LIN {X 0,Y 228.814,Z 416.35,A -85,B 0,C 180,E1 -20899.749,E2 -20899.749} C_VEL
LIN {X 0,Y 233.33,Z 413.266,A -85,B 0,C 180,E1 -20902.12,E2 -20902.12} C_VEL
LIN {X 0,Y 238.29,Z 408.992,A -85,B 0,C 180,E1 -20904.39,E2 -20904.39} C_VEL
LIN {X 0,Y 239.683,Z 407.452,A -85,B 0,C 180,E1 -20905.163,E2 -20905.163} C_VEL
LIN {X 0,Y 241.807,Z 403.361,A -85,B 0,C 180,E1 -20907.714,E2 -20907.714} C_VEL
LIN {X 0,Y 243.168,Z 399.95,A -85,B 0,C 180,E1 -20909.882,E2 -20909.882} C_VEL
LIN {X 0,Y 244.629,Z 395.449,A -85,B 0,C 180,E1 -20913.085,E2 -20913.085} C_VEL
LIN {X 0,Y 245.074,Z 393.5,A -85,B 0,C 180,E1 -20915,E2 -20915} C_VEL
LIN {X 0,Y 245.23,Z 392.181,A -85,B 0,C 180,E1 -20917.004,E2 -20917.004} C_VEL
LIN {X 0,Y 245.282,Z 391.515,A -85,B 0,C 180,E1 -20919.319,E2 -20919.319} C_VEL
LIN {X 0,Y 245.496,Z 391.651,A -85,B 0,C 180,E1 -20921.899,E2 -20921.899} C_VEL
LIN {X 0,Y 245.947,Z 392.643,A -85,B 0,C 180,E1 -20924.407,E2 -20924.407} C_VEL
LIN {X 0,Y 246.92,Z 395.234,A -85,B 0,C 180,E1 -20927.736,E2 -20927.736} C_VEL
LIN {X 0,Y 247.592,Z 398.254,A -85,B 0,C 180,E1 -20930.035,E2 -20930.035} C_VEL
LIN {X 0,Y 247.879,Z 400.529,A -85,B 0,C 180,E1 -20931.409,E2 -20931.409} C_VEL
LIN {X 0,Y 247.014,Z 403.447,A -85,B 0,C 180,E1 -20932.402,E2 -20932.402} C_VEL
LIN {X 0,Y 243.965,Z 411.2,A -85,B 0,C 180,E1 -20934.82,E2 -20934.82} C_VEL
LIN {X 0,Y 240.711,Z 417.71,A -85,B 0,C 180,E1 -20936.808,E2 -20936.808} C_VEL
LIN {X 0,Y 236.558,Z 423.872,A -85,B 0,C 180,E1 -20938.673,E2 -20938.673} C_VEL
LIN {X 0,Y 231.251,Z 430.368,A -85,B 0,C 180,E1 -20940.905,E2 -20940.905} C_VEL
LIN {X 0,Y 225.202,Z 437.275,A -85,B 0,C 180,E1 -20944.093,E2 -20944.093} C_VEL
LIN {X 0,Y 222.213,Z 440.446,A -85,B 0,C 180,E1 -20946.02,E2 -20946.02} C_VEL
LIN {X 0,Y 219.813,Z 442.378,A -85,B 0,C 180,E1 -20947.335,E2 -20947.335} C_VEL
LIN {X 0,Y 214.43,Z 444.919,A -85,B 0,C 180,E1 -20949.437,E2 -20949.437} C_VEL
LIN {X 0,Y 209.432,Z 446.66,A -85,B 0,C 180,E1 -20951.695,E2 -20951.695} C_VEL
LIN {X 0,Y 207.679,Z 447.347,A -85,B 0,C 180,E1 -20953.224,E2 -20953.224} C_VEL
LIN {X 0,Y 206.133,Z 448.199,A -85,B 0,C 180,E1 -20956.192,E2 -20956.192} C_VEL
LIN {X 0,Y 205.327,Z 448.115,A -85,B 0,C 180,E1 -20960.146,E2 -20960.146} C_VEL
LIN {X 0,Y 205.557,Z 446.587,A -85,B 0,C 180,E1 -20964.113,E2 -20964.113} C_VEL
LIN {X 0,Y 206.007,Z 445.284,A -85,B 0,C 180,E1 -20966.088,E2 -20966.088} C_VEL
LIN {X 0,Y 206.791,Z 442.454,A -85,B 0,C 180,E1 -20969.026,E2 -20969.026} C_VEL
LIN {X 0,Y 207.458,Z 438.737,A -85,B 0,C 180,E1 -20971.881,E2 -20971.881} C_VEL
LIN {X 0,Y 206.568,Z 441.761,A -85,B 0,C 180,E1 -20973.902,E2 -20973.902} C_VEL
LIN {X 0,Y 205.939,Z 443.935,A -85,B 0,C 180,E1 -20975.876,E2 -20975.876} C_VEL
LIN {X 0,Y 205.61,Z 445.513,A -85,B 0,C 180,E1 -20977.858,E2 -20977.858} C_VEL
LIN {X 0,Y 205.582,Z 446.527,A -85,B 0,C 180,E1 -20979.842,E2 -20979.842} C_VEL
LIN {X 0,Y 205.912,Z 446.997,A -85,B 0,C 180,E1 -20981.817,E2 -20981.817} C_VEL
LIN {X 0,Y 206.627,Z 446.963,A -85,B 0,C 180,E1 -20983.774,E2 -20983.774} C_VEL
LIN {X 0,Y 207.622,Z 446.402,A -85,B 0,C 180,E1 -20985.712,E2 -20985.712} C_VEL
LIN {X 0,Y 209.104,Z 445.335,A -85,B 0,C 180,E1 -20987.607,E2 -20987.607} C_VEL
LIN {X 0,Y 211.961,Z 442.735,A -85,B 0,C 180,E1 -20990.374,E2 -20990.374} C_VEL
LIN {X 0,Y 215.478,Z 438.804,A -85,B 0,C 180,E1 -20993.041,E2 -20993.041} C_VEL
LIN {X 0,Y 219.824,Z 433.439,A -85,B 0,C 180,E1 -20995.57,E2 -20995.57} C_VEL
LIN {X 0,Y 223.914,Z 427.641,A -85,B 0,C 180,E1 -20997.578,E2 -20997.578} C_VEL
LIN {X 0,Y 228.592,Z 420.356,A -85,B 0,C 180,E1 -20999.467,E2 -20999.467} C_VEL
LIN {X 0,Y 232.382,Z 412.031,A -85,B 0,C 180,E1 -21001.4,E2 -21001.4} C_VEL
LIN {X 0,Y 233.877,Z 408.212,A -85,B 0,C 180,E1 -21002.188,E2 -21002.188} C_VEL
LIN {X 0,Y 235.674,Z 399.15,A -85,B 0,C 180,E1 -21004.513,E2 -21004.513} C_VEL
LIN {X 0,Y 236.749,Z 389.553,A -85,B 0,C 180,E1 -21007.182,E2 -21007.182} C_VEL
LIN {X 0,Y 236.748,Z 388.634,A -85,B 0,C 180,E1 -21007.486,E2 -21007.486} C_VEL
LIN {X 0,Y 236.034,Z 385.627,A -85,B 0,C 180,E1 -21009.268,E2 -21009.268} C_VEL
LIN {X 0,Y 235.075,Z 383.096,A -85,B 0,C 180,E1 -21011.63,E2 -21011.63} C_VEL
LIN {X 0,Y 234.344,Z 381.808,A -85,B 0,C 180,E1 -21013.963,E2 -21013.963} C_VEL
LIN {X 0,Y 233.881,Z 381.582,A -85,B 0,C 180,E1 -21016.277,E2 -21016.277} C_VEL
LIN {X 0,Y 233.809,Z 382.151,A -85,B 0,C 180,E1 -21018.718,E2 -21018.718} C_VEL
LIN {X 0,Y 234.028,Z 383.771,A -85,B 0,C 180,E1 -21021.334,E2 -21021.334} C_VEL
LIN {X 0,Y 234.447,Z 385.325,A -85,B 0,C 180,E1 -21023.161,E2 -21023.161} C_VEL
LIN {X 0,Y 234.718,Z 388.125,A -85,B 0,C 180,E1 -21025.324,E2 -21025.324} C_VEL
LIN {X 0,Y 234.45,Z 392.693,A -85,B 0,C 180,E1 -21027.833,E2 -21027.833} C_VEL
LIN {X 0,Y 233.699,Z 398.365,A -85,B 0,C 180,E1 -21030.705,E2 -21030.705} C_VEL
LIN {X 0,Y 232.609,Z 403.003,A -85,B 0,C 180,E1 -21033.048,E2 -21033.048} C_VEL
LIN {X 0,Y 231.392,Z 406.408,A -85,B 0,C 180,E1 -21034.833,E2 -21034.833} C_VEL
LIN {X 0,Y 230.175,Z 408.313,A -85,B 0,C 180,E1 -21035.655,E2 -21035.655} C_VEL
LIN {X 0,Y 225.28,Z 413.35,A -85,B 0,C 180,E1 -21038.013,E2 -21038.013} C_VEL
LIN {X 0,Y 222.294,Z 415.749,A -85,B 0,C 180,E1 -21039.647,E2 -21039.647} C_VEL
LIN {X 0,Y 219.533,Z 417.471,A -85,B 0,C 180,E1 -21041.327,E2 -21041.327} C_VEL
LIN {X 0,Y 216.997,Z 418.533,A -85,B 0,C 180,E1 -21043.051,E2 -21043.051} C_VEL
LIN {X 0,Y 214.633,Z 418.98,A -85,B 0,C 180,E1 -21044.812,E2 -21044.812} C_VEL
LIN {X 0,Y 212.473,Z 418.818,A -85,B 0,C 180,E1 -21046.61,E2 -21046.61} C_VEL
LIN {X 0,Y 210.527,Z 418.027,A -85,B 0,C 180,E1 -21048.443,E2 -21048.443} C_VEL
LIN {X 0,Y 208.193,Z 415.631,A -85,B 0,C 180,E1 -21051.26,E2 -21051.26} C_VEL
LIN {X 0,Y 206.472,Z 411.79,A -85,B 0,C 180,E1 -21054.137,E2 -21054.137} C_VEL
LIN {X 0,Y 205.572,Z 406.34,A -85,B 0,C 180,E1 -21057.058,E2 -21057.058} C_VEL
LIN {X 0,Y 205.271,Z 400.286,A -85,B 0,C 180,E1 -21059.507,E2 -21059.507} C_VEL
LIN {X 0,Y 205.338,Z 392.617,A -85,B 0,C 180,E1 -21061.959,E2 -21061.959} C_VEL
LIN {X 0,Y 205.793,Z 383.712,A -85,B 0,C 180,E1 -21064.159,E2 -21064.159} C_VEL
LIN {X 0,Y 206.062,Z 376.071,A -85,B 0,C 180,E1 -21065.625,E2 -21065.625} C_VEL
LIN {X 0,Y 206.367,Z 365.456,A -85,B 0,C 180,E1 -21067.212,E2 -21067.212} C_VEL
LIN {X 0,Y 206.597,Z 356.563,A -85,B 0,C 180,E1 -21068.221,E2 -21068.221} C_VEL
LIN {X 0,Y 205.887,Z 341.814,A -85,B 0,C 180,E1 -21076.475,E2 -21076.475} C_VEL
LIN {X 0,Y 206.128,Z 333.911,A -85,B 0,C 180,E1 -21080.975,E2 -21080.975} C_VEL
LIN {X 0,Y 206.537,Z 324.736,A -85,B 0,C 180,E1 -21086.252,E2 -21086.252} C_VEL
LIN {X 0,Y 206.884,Z 318.714,A -85,B 0,C 180,E1 -21089.787,E2 -21089.787} C_VEL
LIN {X 0,Y 206.754,Z 318.73,A -85,B 0,C 180,E1 -21092.944,E2 -21092.944} C_VEL
LIN {X 0,Y 206.669,Z 318.74,A -85,B 0,C 180,E1 -21097.739,E2 -21097.739} C_VEL
LIN {X 0,Y 206.628,Z 318.743,A -85,B 0,C 180,E1 -21101.558,E2 -21101.558} C_VEL
LIN {X 0,Y 206.624,Z 318.746,A -85,B 0,C 180,E1 -21105.58,E2 -21105.58} C_VEL
LIN {X 0,Y 206.652,Z 318.74,A -85,B 0,C 180,E1 -21109.747,E2 -21109.747} C_VEL
LIN {X 0,Y 206.691,Z 318.739,A -85,B 0,C 180,E1 -21114.687,E2 -21114.687} C_VEL
LIN {X 0,Y 206.714,Z 318.731,A -85,B 0,C 180,E1 -21119.337,E2 -21119.337} C_VEL
LIN {X 0,Y 206.724,Z 318.733,A -85,B 0,C 180,E1 -21123.771,E2 -21123.771} C_VEL
LIN {X 0,Y 206.749,Z 318.728,A -85,B 0,C 180,E1 -21128.042,E2 -21128.042} C_VEL
LIN {X 0,Y 206.867,Z 318.717,A -85,B 0,C 180,E1 -21132.196,E2 -21132.196} C_VEL
LIN {X 0,Y 206.88,Z 318.713,A -85,B 0,C 180,E1 -21136.243,E2 -21136.243} C_VEL
LIN {X 0,Y 207.069,Z 318.693,A -85,B 0,C 180,E1 -21140.229,E2 -21140.229} C_VEL
LIN {X 0,Y 207.029,Z 318.695,A -85,B 0,C 180,E1 -21144.155,E2 -21144.155} C_VEL
LIN {X 0,Y 207.334,Z 318.659,A -85,B 0,C 180,E1 -21148.057,E2 -21148.057} C_VEL
LIN {X 0,Y 207.469,Z 318.644,A -85,B 0,C 180,E1 -21150,E2 -21150} C_VEL
LIN {X 0,Y 207.334,Z 318.659,A -85,B 0,C 180,E1 -21151.943,E2 -21151.943} C_VEL
LIN {X 0,Y 207.118,Z 318.687,A -85,B 0,C 180,E1 -21157.801,E2 -21157.801} C_VEL
LIN {X 0,Y 206.91,Z 318.709,A -85,B 0,C 180,E1 -21161.759,E2 -21161.759} C_VEL
LIN {X 0,Y 206.855,Z 318.719,A -85,B 0,C 180,E1 -21165.772,E2 -21165.772} C_VEL
LIN {X 0,Y 206.803,Z 318.722,A -85,B 0,C 180,E1 -21169.867,E2 -21169.867} C_VEL
LIN {X 0,Y 206.759,Z 318.729,A -85,B 0,C 180,E1 -21174.073,E2 -21174.073} C_VEL
LIN {X 0,Y 206.735,Z 318.73,A -85,B 0,C 180,E1 -21178.42,E2 -21178.42} C_VEL
LIN {X 0,Y 206.694,Z 318.737,A -85,B 0,C 180,E1 -21182.959,E2 -21182.959} C_VEL
LIN {X 0,Y 206.672,Z 318.737,A -85,B 0,C 180,E1 -21187.742,E2 -21187.742} C_VEL
LIN {X 0,Y 206.633,Z 318.745,A -85,B 0,C 180,E1 -21191.564,E2 -21191.564} C_VEL
LIN {X 0,Y 206.624,Z 318.744,A -85,B 0,C 180,E1 -21195.585,E2 -21195.585} C_VEL
LIN {X 0,Y 206.647,Z 318.742,A -85,B 0,C 180,E1 -21199.749,E2 -21199.749} C_VEL
LIN {X 0,Y 206.783,Z 318.725,A -85,B 0,C 180,E1 -21204.709,E2 -21204.709} C_VEL
LIN {X 0,Y 207.122,Z 318.815,A -85,B 0,C 180,E1 -21208.351,E2 -21208.351} C_VEL
LIN {X 0,Y 206.657,Z 323.186,A -85,B 0,C 180,E1 -21212.155,E2 -21212.155} C_VEL
LIN {X 0,Y 206.05,Z 328.932,A -85,B 0,C 180,E1 -21217.062,E2 -21217.062} C_VEL
LIN {X 0,Y 205.493,Z 334.922,A -85,B 0,C 180,E1 -21222.076,E2 -21222.076} C_VEL
LIN {X 0,Y 205.269,Z 341.862,A -85,B 0,C 180,E1 -21227.709,E2 -21227.709} C_VEL
LIN {X 0,Y 206.4,Z 354.238,A -85,B 0,C 180,E1 -21229.085,E2 -21229.085} C_VEL
LIN {X 0,Y 206.727,Z 360.644,A -85,B 0,C 180,E1 -21229.969,E2 -21229.969} C_VEL
LIN {X 0,Y 206.197,Z 372.124,A -85,B 0,C 180,E1 -21231.924,E2 -21231.924} C_VEL
LIN {X 0,Y 205.81,Z 382.31,A -85,B 0,C 180,E1 -21234.123,E2 -21234.123} C_VEL
LIN {X 0,Y 205.337,Z 391.3,A -85,B 0,C 180,E1 -21236.569,E2 -21236.569} C_VEL
LIN {X 0,Y 205.133,Z 399.93,A -85,B 0,C 180,E1 -21239.512,E2 -21239.512} C_VEL
LIN {X 0,Y 205.32,Z 405.672,A -85,B 0,C 180,E1 -21241.964,E2 -21241.964} C_VEL
LIN {X 0,Y 206.134,Z 411.087,A -85,B 0,C 180,E1 -21244.892,E2 -21244.892} C_VEL
LIN {X 0,Y 207.525,Z 415.168,A -85,B 0,C 180,E1 -21247.788,E2 -21247.788} C_VEL
LIN {X 0,Y 208.827,Z 417.148,A -85,B 0,C 180,E1 -21249.69,E2 -21249.69} C_VEL
LIN {X 0,Y 210.385,Z 418.6,A -85,B 0,C 180,E1 -21251.565,E2 -21251.565} C_VEL
LIN {X 0,Y 212.31,Z 419.539,A -85,B 0,C 180,E1 -21253.401,E2 -21253.401} C_VEL
LIN {X 0,Y 214.482,Z 419.914,A -85,B 0,C 180,E1 -21255.199,E2 -21255.199} C_VEL
LIN {X 0,Y 216.874,Z 419.813,A -85,B 0,C 180,E1 -21256.959,E2 -21256.959} C_VEL
LIN {X 0,Y 219.491,Z 419.201,A -85,B 0,C 180,E1 -21258.677,E2 -21258.677} C_VEL
LIN {X 0,Y 222.323,Z 418.076,A -85,B 0,C 180,E1 -21260.351,E2 -21260.351} C_VEL
LIN {X 0,Y 227.004,Z 415.473,A -85,B 0,C 180,E1 -21262.77,E2 -21262.77} C_VEL
LIN {X 0,Y 232.143,Z 411.656,A -85,B 0,C 180,E1 -21265.08,E2 -21265.08} C_VEL
LIN {X 0,Y 233.739,Z 410.198,A -85,B 0,C 180,E1 -21265.85,E2 -21265.85} C_VEL
LIN {X 0,Y 236.189,Z 406.575,A -85,B 0,C 180,E1 -21268.433,E2 -21268.433} C_VEL
LIN {X 0,Y 238.124,Z 402.905,A -85,B 0,C 180,E1 -21271.139,E2 -21271.139} C_VEL
LIN {X 0,Y 239.643,Z 399.623,A -85,B 0,C 180,E1 -21273.865,E2 -21273.865} C_VEL
LIN {X 0,Y 240.137,Z 398.024,A -85,B 0,C 180,E1 -21275.829,E2 -21275.829} C_VEL
LIN {X 0,Y 240.368,Z 397.115,A -85,B 0,C 180,E1 -21277.882,E2 -21277.882} C_VEL
LIN {X 0,Y 240.641,Z 396.83,A -85,B 0,C 180,E1 -21280.594,E2 -21280.594} C_VEL
LIN {X 0,Y 241.068,Z 397.401,A -85,B 0,C 180,E1 -21283.211,E2 -21283.211} C_VEL
LIN {X 0,Y 241.771,Z 399.583,A -85,B 0,C 180,E1 -21286.615,E2 -21286.615} C_VEL
LIN {X 0,Y 242.392,Z 401.958,A -85,B 0,C 180,E1 -21288.928,E2 -21288.928} C_VEL
LIN {X 0,Y 242.593,Z 404.996,A -85,B 0,C 180,E1 -21290.942,E2 -21290.942} C_VEL
LIN {X 0,Y 239.242,Z 412.361,A -85,B 0,C 180,E1 -21293.461,E2 -21293.461} C_VEL
LIN {X 0,Y 235.819,Z 418.507,A -85,B 0,C 180,E1 -21295.511,E2 -21295.511} C_VEL
LIN {X 0,Y 231.575,Z 424.327,A -85,B 0,C 180,E1 -21297.405,E2 -21297.405} C_VEL
LIN {X 0,Y 225.149,Z 431.45,A -85,B 0,C 180,E1 -21300.037,E2 -21300.037} C_VEL
LIN {X 0,Y 218.862,Z 437.795,A -85,B 0,C 180,E1 -21303.284,E2 -21303.284} C_VEL
LIN {X 0,Y 214.916,Z 441.499,A -85,B 0,C 180,E1 -21305.873,E2 -21305.873} C_VEL
LIN {X 0,Y 211.597,Z 444.363,A -85,B 0,C 180,E1 -21308.57,E2 -21308.57} C_VEL
LIN {X 0,Y 208.267,Z 446.981,A -85,B 0,C 180,E1 -21312.32,E2 -21312.32} C_VEL
LIN {X 0,Y 207.679,Z 447.347,A -85,B 0,C 180,E1 -21313.224,E2 -21313.224} C_VEL
LIN {X 0,Y 206.148,Z 447.868,A -85,B 0,C 180,E1 -21314.798,E2 -21314.798} C_VEL
LIN {X 0,Y 202.33,Z 447.811,A -85,B 0,C 180,E1 -21317.362,E2 -21317.362} C_VEL
LIN {X 0,Y 199.528,Z 447.131,A -85,B 0,C 180,E1 -21319.475,E2 -21319.475} C_VEL
LIN {X 0,Y 198.409,Z 446.41,A -85,B 0,C 180,E1 -21321.137,E2 -21321.137} C_VEL
LIN {X 0,Y 198.339,Z 446.162,A -85,B 0,C 180,E1 -21321.704,E2 -21321.704} C_VEL
LIN {X 0,Y 198.614,Z 445.033,A -85,B 0,C 180,E1 -21323.906,E2 -21323.906} C_VEL
LIN {X 0,Y 199.111,Z 443.561,A -85,B 0,C 180,E1 -21325.952,E2 -21325.952} C_VEL
LIN {X 0,Y 199.963,Z 440.509,A -85,B 0,C 180,E1 -21328.993,E2 -21328.993} C_VEL
LIN {X 0,Y 200.762,Z 436.383,A -85,B 0,C 180,E1 -21331.943,E2 -21331.943} C_VEL
LIN {X 0,Y 199.397,Z 440.916,A -85,B 0,C 180,E1 -21335.055,E2 -21335.055} C_VEL
LIN {X 0,Y 198.738,Z 443.853,A -85,B 0,C 180,E1 -21338.132,E2 -21338.132} C_VEL
LIN {X 0,Y 198.696,Z 445.101,A -85,B 0,C 180,E1 -21340.187,E2 -21340.187} C_VEL
LIN {X 0,Y 199.013,Z 445.841,A -85,B 0,C 180,E1 -21342.233,E2 -21342.233} C_VEL
LIN {X 0,Y 199.745,Z 446.071,A -85,B 0,C 180,E1 -21344.258,E2 -21344.258} C_VEL
LIN {X 0,Y 200.795,Z 445.783,A -85,B 0,C 180,E1 -21346.261,E2 -21346.261} C_VEL
LIN {X 0,Y 202.349,Z 444.989,A -85,B 0,C 180,E1 -21348.215,E2 -21348.215} C_VEL
LIN {X 0,Y 204.237,Z 443.668,A -85,B 0,C 180,E1 -21350.128,E2 -21350.128} C_VEL
LIN {X 0,Y 207.729,Z 440.671,A -85,B 0,C 180,E1 -21352.897,E2 -21352.897} C_VEL
LIN {X 0,Y 211.919,Z 436.396,A -85,B 0,C 180,E1 -21355.539,E2 -21355.539} C_VEL
LIN {X 0,Y 216.855,Z 430.572,A -85,B 0,C 180,E1 -21358.03,E2 -21358.03} C_VEL
LIN {X 0,Y 221.573,Z 424.413,A -85,B 0,C 180,E1 -21359.972,E2 -21359.972} C_VEL
LIN {X 0,Y 225.339,Z 418.46,A -85,B 0,C 180,E1 -21361.494,E2 -21361.494} C_VEL
LIN {X 0,Y 228.541,Z 411.982,A -85,B 0,C 180,E1 -21363.034,E2 -21363.034} C_VEL
LIN {X 0,Y 230.325,Z 406.43,A -85,B 0,C 180,E1 -21364.524,E2 -21364.524} C_VEL
LIN {X 0,Y 231.714,Z 400.773,A -85,B 0,C 180,E1 -21366.139,E2 -21366.139} C_VEL
LIN {X 0,Y 232.872,Z 394.863,A -85,B 0,C 180,E1 -21367.909,E2 -21367.909} C_VEL
LIN {X 0,Y 232.978,Z 393.711,A -85,B 0,C 180,E1 -21368.34,E2 -21368.34} C_VEL
LIN {X 0,Y 232.682,Z 392.043,A -85,B 0,C 180,E1 -21369.368,E2 -21369.368} C_VEL
LIN {X 0,Y 232.231,Z 390.265,A -85,B 0,C 180,E1 -21370.834,E2 -21370.834} C_VEL
LIN {X 0,Y 231.445,Z 388.58,A -85,B 0,C 180,E1 -21373.213,E2 -21373.213} C_VEL
LIN {X 0,Y 230.844,Z 387.995,A -85,B 0,C 180,E1 -21375.552,E2 -21375.552} C_VEL
LIN {X 0,Y 230.526,Z 388.25,A -85,B 0,C 180,E1 -21377.876,E2 -21377.876} C_VEL
LIN {X 0,Y 230.45,Z 389.223,A -85,B 0,C 180,E1 -21380.173,E2 -21380.173} C_VEL
LIN {X 0,Y 230.592,Z 391.857,A -85,B 0,C 180,E1 -21383.532,E2 -21383.532} C_VEL
LIN {X 0,Y 230.371,Z 394.396,A -85,B 0,C 180,E1 -21385.457,E2 -21385.457} C_VEL
LIN {X 0,Y 229.212,Z 399.768,A -85,B 0,C 180,E1 -21388.582,E2 -21388.582} C_VEL
LIN {X 0,Y 227.761,Z 404.5,A -85,B 0,C 180,E1 -21391.242,E2 -21391.242} C_VEL
LIN {X 0,Y 225.548,Z 409.487,A -85,B 0,C 180,E1 -21394.134,E2 -21394.134} C_VEL
LIN {X 0,Y 222.282,Z 412.838,A -85,B 0,C 180,E1 -21395.728,E2 -21395.728} C_VEL
LIN {X 0,Y 217.399,Z 416.723,A -85,B 0,C 180,E1 -21398.173,E2 -21398.173} C_VEL
LIN {X 0,Y 212.968,Z 418.983,A -85,B 0,C 180,E1 -21400.729,E2 -21400.729} C_VEL
LIN {X 0,Y 210.317,Z 419.73,A -85,B 0,C 180,E1 -21402.495,E2 -21402.495} C_VEL
LIN {X 0,Y 207.848,Z 419.882,A -85,B 0,C 180,E1 -21404.303,E2 -21404.303} C_VEL
LIN {X 0,Y 205.589,Z 419.417,A -85,B 0,C 180,E1 -21406.153,E2 -21406.153} C_VEL
LIN {X 0,Y 203.585,Z 418.333,A -85,B 0,C 180,E1 -21408.043,E2 -21408.043} C_VEL
LIN {X 0,Y 201.187,Z 415.557,A -85,B 0,C 180,E1 -21410.953,E2 -21410.953} C_VEL
LIN {X 0,Y 199.424,Z 411.239,A -85,B 0,C 180,E1 -21413.929,E2 -21413.929} C_VEL
LIN {X 0,Y 198.636,Z 406.411,A -85,B 0,C 180,E1 -21416.448,E2 -21416.448} C_VEL
LIN {X 0,Y 198.291,Z 400.173,A -85,B 0,C 180,E1 -21418.982,E2 -21418.982} C_VEL
LIN {X 0,Y 198.369,Z 392.244,A -85,B 0,C 180,E1 -21421.52,E2 -21421.52} C_VEL
LIN {X 0,Y 198.8,Z 383.191,A -85,B 0,C 180,E1 -21423.798,E2 -21423.798} C_VEL
LIN {X 0,Y 199.056,Z 376.824,A -85,B 0,C 180,E1 -21425.061,E2 -21425.061} C_VEL
LIN {X 0,Y 199.344,Z 366.227,A -85,B 0,C 180,E1 -21426.704,E2 -21426.704} C_VEL
LIN {X 0,Y 199.593,Z 357.24,A -85,B 0,C 180,E1 -21427.776,E2 -21427.776} C_VEL
LIN {X 0,Y 198.807,Z 342.107,A -85,B 0,C 180,E1 -21436.425,E2 -21436.425} C_VEL
LIN {X 0,Y 199.075,Z 332.935,A -85,B 0,C 180,E1 -21441.755,E2 -21441.755} C_VEL
LIN {X 0,Y 199.442,Z 325.467,A -85,B 0,C 180,E1 -21446.131,E2 -21446.131} C_VEL
LIN {X 0,Y 199.773,Z 319.601,A -85,B 0,C 180,E1 -21449.648,E2 -21449.648} C_VEL
LIN {X 0,Y 199.949,Z 319.577,A -85,B 0,C 180,E1 -21450.638,E2 -21450.638} C_VEL
LIN {X 0,Y 199.6,Z 319.62,A -85,B 0,C 180,E1 -21456.764,E2 -21456.764} C_VEL
LIN {X 0,Y 199.592,Z 319.623,A -85,B 0,C 180,E1 -21459.328,E2 -21459.328} C_VEL
LIN {X 0,Y 199.562,Z 319.622,A -85,B 0,C 180,E1 -21462.306,E2 -21462.306} C_VEL
LIN {X 0,Y 199.57,Z 319.626,A -85,B 0,C 180,E1 -21465.226,E2 -21465.226} C_VEL
LIN {X 0,Y 199.57,Z 319.624,A -85,B 0,C 180,E1 -21468.002,E2 -21468.002} C_VEL
LIN {X 0,Y 199.603,Z 319.619,A -85,B 0,C 180,E1 -21470.766,E2 -21470.766} C_VEL
LIN {X 0,Y 199.605,Z 319.62,A -85,B 0,C 180,E1 -21475.712,E2 -21475.712} C_VEL
LIN {X 0,Y 199.692,Z 319.609,A -85,B 0,C 180,E1 -21478.135,E2 -21478.135} C_VEL
LIN {X 0,Y 199.679,Z 319.613,A -85,B 0,C 180,E1 -21482.77,E2 -21482.77} C_VEL
LIN {X 0,Y 199.729,Z 319.602,A -85,B 0,C 180,E1 -21487.228,E2 -21487.228} C_VEL
LIN {X 0,Y 199.828,Z 319.592,A -85,B 0,C 180,E1 -21491.721,E2 -21491.721} C_VEL
LIN {X 0,Y 199.822,Z 319.592,A -85,B 0,C 180,E1 -21495.747,E2 -21495.747} C_VEL
LIN {X 0,Y 200.012,Z 319.569,A -85,B 0,C 180,E1 -21499.881,E2 -21499.881} C_VEL
LIN {X 0,Y 199.993,Z 319.573,A -85,B 0,C 180,E1 -21503.948,E2 -21503.948} C_VEL
LIN {X 0,Y 200.276,Z 319.537,A -85,B 0,C 180,E1 -21507.989,E2 -21507.989} C_VEL
LIN {X 0,Y 200.436,Z 319.52,A -85,B 0,C 180,E1 -21510,E2 -21510} C_VEL
LIN {X 0,Y 199.982,Z 319.571,A -85,B 0,C 180,E1 -21514.03,E2 -21514.03} C_VEL
LIN {X 0,Y 200.066,Z 319.564,A -85,B 0,C 180,E1 -21518.078,E2 -21518.078} C_VEL
LIN {X 0,Y 199.861,Z 319.585,A -85,B 0,C 180,E1 -21522.18,E2 -21522.18} C_VEL
LIN {X 0,Y 199.795,Z 319.596,A -85,B 0,C 180,E1 -21526.344,E2 -21526.344} C_VEL
LIN {X 0,Y 199.732,Z 319.601,A -85,B 0,C 180,E1 -21530.602,E2 -21530.602} C_VEL
LIN {X 0,Y 199.667,Z 319.613,A -85,B 0,C 180,E1 -21534.985,E2 -21534.985} C_VEL
LIN {X 0,Y 199.666,Z 319.61,A -85,B 0,C 180,E1 -21539.524,E2 -21539.524} C_VEL
LIN {X 0,Y 199.669,Z 319.611,A -85,B 0,C 180,E1 -21542.36,E2 -21542.36} C_VEL
LIN {X 0,Y 199.615,Z 319.619,A -85,B 0,C 180,E1 -21546.765,E2 -21546.765} C_VEL
LIN {X 0,Y 199.6,Z 319.62,A -85,B 0,C 180,E1 -21549.33,E2 -21549.33} C_VEL
LIN {X 0,Y 199.565,Z 319.625,A -85,B 0,C 180,E1 -21552.312,E2 -21552.312} C_VEL
LIN {X 0,Y 199.57,Z 319.624,A -85,B 0,C 180,E1 -21555.23,E2 -21555.23} C_VEL
LIN {X 0,Y 199.566,Z 319.621,A -85,B 0,C 180,E1 -21558.006,E2 -21558.006} C_VEL
LIN {X 0,Y 199.603,Z 319.622,A -85,B 0,C 180,E1 -21560.771,E2 -21560.771} C_VEL
LIN {X 0,Y 199.811,Z 319.59,A -85,B 0,C 180,E1 -21565.756,E2 -21565.756} C_VEL
LIN {X 0,Y 200.078,Z 319.751,A -85,B 0,C 180,E1 -21568.503,E2 -21568.503} C_VEL
LIN {X 0,Y 199.478,Z 324.503,A -85,B 0,C 180,E1 -21572.744,E2 -21572.744} C_VEL
LIN {X 0,Y 198.959,Z 329.519,A -85,B 0,C 180,E1 -21577.138,E2 -21577.138} C_VEL
LIN {X 0,Y 198.464,Z 334.486,A -85,B 0,C 180,E1 -21581.418,E2 -21581.418} C_VEL
LIN {X 0,Y 198.173,Z 342.075,A -85,B 0,C 180,E1 -21587.847,E2 -21587.847} C_VEL
LIN {X 0,Y 199.381,Z 354.911,A -85,B 0,C 180,E1 -21589.338,E2 -21589.338} C_VEL
LIN {X 0,Y 199.679,Z 359.972,A -85,B 0,C 180,E1 -21590.056,E2 -21590.056} C_VEL
LIN {X 0,Y 199.134,Z 371.832,A -85,B 0,C 180,E1 -21592.142,E2 -21592.142} C_VEL
LIN {X 0,Y 198.764,Z 382.122,A -85,B 0,C 180,E1 -21594.423,E2 -21594.423} C_VEL
LIN {X 0,Y 198.286,Z 391.281,A -85,B 0,C 180,E1 -21596.955,E2 -21596.955} C_VEL
LIN {X 0,Y 198.098,Z 398.717,A -85,B 0,C 180,E1 -21599.494,E2 -21599.494} C_VEL
LIN {X 0,Y 198.379,Z 405.836,A -85,B 0,C 180,E1 -21602.541,E2 -21602.541} C_VEL
LIN {X 0,Y 199.07,Z 410.594,A -85,B 0,C 180,E1 -21605.066,E2 -21605.066} C_VEL
LIN {X 0,Y 200.492,Z 415.01,A -85,B 0,C 180,E1 -21608.063,E2 -21608.063} C_VEL
LIN {X 0,Y 201.831,Z 417.25,A -85,B 0,C 180,E1 -21610.029,E2 -21610.029} C_VEL
LIN {X 0,Y 203.454,Z 418.936,A -85,B 0,C 180,E1 -21611.964,E2 -21611.964} C_VEL
LIN {X 0,Y 205.43,Z 420.117,A -85,B 0,C 180,E1 -21613.858,E2 -21613.858} C_VEL
LIN {X 0,Y 207.678,Z 420.768,A -85,B 0,C 180,E1 -21615.71,E2 -21615.71} C_VEL
LIN {X 0,Y 210.159,Z 420.904,A -85,B 0,C 180,E1 -21617.518,E2 -21617.518} C_VEL
LIN {X 0,Y 212.88,Z 420.565,A -85,B 0,C 180,E1 -21619.28,E2 -21619.28} C_VEL
LIN {X 0,Y 215.839,Z 419.711,A -85,B 0,C 180,E1 -21620.99,E2 -21620.99} C_VEL
LIN {X 0,Y 218.986,Z 418.408,A -85,B 0,C 180,E1 -21622.654,E2 -21622.654} C_VEL
LIN {X 0,Y 224.198,Z 415.421,A -85,B 0,C 180,E1 -21625.038,E2 -21625.038} C_VEL
LIN {X 0,Y 227.769,Z 412.903,A -85,B 0,C 180,E1 -21626.58,E2 -21626.58} C_VEL
LIN {X 0,Y 229.724,Z 410.725,A -85,B 0,C 180,E1 -21628.309,E2 -21628.309} C_VEL
LIN {X 0,Y 232.072,Z 407.517,A -85,B 0,C 180,E1 -21630.988,E2 -21630.988} C_VEL
LIN {X 0,Y 233.385,Z 405.461,A -85,B 0,C 180,E1 -21632.825,E2 -21632.825} C_VEL
LIN {X 0,Y 234.478,Z 403.658,A -85,B 0,C 180,E1 -21634.717,E2 -21634.717} C_VEL
LIN {X 0,Y 235.048,Z 402.512,A -85,B 0,C 180,E1 -21636.729,E2 -21636.729} C_VEL
LIN {X 0,Y 235.414,Z 401.944,A -85,B 0,C 180,E1 -21639.086,E2 -21639.086} C_VEL
LIN {X 0,Y 235.844,Z 402.099,A -85,B 0,C 180,E1 -21641.842,E2 -21641.842} C_VEL
LIN {X 0,Y 236.313,Z 403.137,A -85,B 0,C 180,E1 -21644.458,E2 -21644.458} C_VEL
LIN {X 0,Y 237.025,Z 405.728,A -85,B 0,C 180,E1 -21647.843,E2 -21647.843} C_VEL
LIN {X 0,Y 237.239,Z 407.46,A -85,B 0,C 180,E1 -21649.327,E2 -21649.327} C_VEL
LIN {X 0,Y 237.026,Z 409.226,A -85,B 0,C 180,E1 -21650.439,E2 -21650.439} C_VEL
LIN {X 0,Y 232.487,Z 417.155,A -85,B 0,C 180,E1 -21653.342,E2 -21653.342} C_VEL
LIN {X 0,Y 228.535,Z 422.709,A -85,B 0,C 180,E1 -21655.325,E2 -21655.325} C_VEL
LIN {X 0,Y 222.787,Z 428.866,A -85,B 0,C 180,E1 -21657.569,E2 -21657.569} C_VEL
LIN {X 0,Y 217.352,Z 434.031,A -85,B 0,C 180,E1 -21659.921,E2 -21659.921} C_VEL
LIN {X 0,Y 211.13,Z 439.474,A -85,B 0,C 180,E1 -21663.296,E2 -21663.296} C_VEL
LIN {X 0,Y 207.213,Z 442.556,A -85,B 0,C 180,E1 -21665.983,E2 -21665.983} C_VEL
LIN {X 0,Y 203.111,Z 445.423,A -85,B 0,C 180,E1 -21669.756,E2 -21669.756} C_VEL
LIN {X 0,Y 200.249,Z 446.996,A -85,B 0,C 180,E1 -21673.694,E2 -21673.694} C_VEL
LIN {X 0,Y 198.669,Z 447.203,A -85,B 0,C 180,E1 -21677.746,E2 -21677.746} C_VEL
LIN {X 0,Y 198.339,Z 446.162,A -85,B 0,C 180,E1 -21681.704,E2 -21681.704} C_VEL
LIN {X 0,Y 197.882,Z 445.227,A -85,B 0,C 180,E1 -21683.386,E2 -21683.386} C_VEL
LIN {X 0,Y 196.723,Z 443.737,A -85,B 0,C 180,E1 -21685.024,E2 -21685.024} C_VEL
LIN {X 0,Y 194.092,Z 439.647,A -85,B 0,C 180,E1 -21688.247,E2 -21688.247} C_VEL
LIN {X 0,Y 193.56,Z 436.466,A -85,B 0,C 180,E1 -21690.415,E2 -21690.415} C_VEL
LIN {X 0,Y 194.095,Z 434.047,A -85,B 0,C 180,E1 -21692.14,E2 -21692.14} C_VEL
LIN {X 0,Y 192.669,Z 438.741,A -85,B 0,C 180,E1 -21695.232,E2 -21695.232} C_VEL
LIN {X 0,Y 191.886,Z 442.139,A -85,B 0,C 180,E1 -21698.532,E2 -21698.532} C_VEL
LIN {X 0,Y 191.848,Z 443.532,A -85,B 0,C 180,E1 -21700.554,E2 -21700.554} C_VEL
LIN {X 0,Y 192.161,Z 444.471,A -85,B 0,C 180,E1 -21702.676,E2 -21702.676} C_VEL
LIN {X 0,Y 192.915,Z 444.942,A -85,B 0,C 180,E1 -21704.774,E2 -21704.774} C_VEL
LIN {X 0,Y 194.012,Z 444.919,A -85,B 0,C 180,E1 -21706.846,E2 -21706.846} C_VEL
LIN {X 0,Y 195.621,Z 444.422,A -85,B 0,C 180,E1 -21708.865,E2 -21708.865} C_VEL
LIN {X 0,Y 197.58,Z 443.419,A -85,B 0,C 180,E1 -21710.837,E2 -21710.837} C_VEL
LIN {X 0,Y 201.21,Z 440.929,A -85,B 0,C 180,E1 -21713.683,E2 -21713.683} C_VEL
LIN {X 0,Y 205.595,Z 437.216,A -85,B 0,C 180,E1 -21716.384,E2 -21716.384} C_VEL
LIN {X 0,Y 210.709,Z 432.085,A -85,B 0,C 180,E1 -21718.923,E2 -21718.923} C_VEL
LIN {X 0,Y 215.579,Z 426.554,A -85,B 0,C 180,E1 -21720.895,E2 -21720.895} C_VEL
LIN {X 0,Y 219.65,Z 421.191,A -85,B 0,C 180,E1 -21722.408,E2 -21722.408} C_VEL
LIN {X 0,Y 224.009,Z 413.694,A -85,B 0,C 180,E1 -21724.384,E2 -21724.384} C_VEL
LIN {X 0,Y 226.286,Z 407.797,A -85,B 0,C 180,E1 -21726.165,E2 -21726.165} C_VEL
LIN {X 0,Y 228.855,Z 399.234,A -85,B 0,C 180,E1 -21728.89,E2 -21728.89} C_VEL
LIN {X 0,Y 228.691,Z 397.254,A -85,B 0,C 180,E1 -21730.193,E2 -21730.193} C_VEL
LIN {X 0,Y 228.016,Z 395.042,A -85,B 0,C 180,E1 -21732.695,E2 -21732.695} C_VEL
LIN {X 0,Y 227.303,Z 394.146,A -85,B 0,C 180,E1 -21735.328,E2 -21735.328} C_VEL
LIN {X 0,Y 226.778,Z 394.395,A -85,B 0,C 180,E1 -21738.054,E2 -21738.054} C_VEL
LIN {X 0,Y 226.332,Z 396.083,A -85,B 0,C 180,E1 -21741.606,E2 -21741.606} C_VEL
LIN {X 0,Y 226.08,Z 398.111,A -85,B 0,C 180,E1 -21743.925,E2 -21743.925} C_VEL
LIN {X 0,Y 225.345,Z 400.753,A -85,B 0,C 180,E1 -21745.846,E2 -21745.846} C_VEL
LIN {X 0,Y 223.719,Z 404.947,A -85,B 0,C 180,E1 -21748.539,E2 -21748.539} C_VEL
LIN {X 0,Y 221.479,Z 409.63,A -85,B 0,C 180,E1 -21751.574,E2 -21751.574} C_VEL
LIN {X 0,Y 219.629,Z 412.342,A -85,B 0,C 180,E1 -21753.383,E2 -21753.383} C_VEL
LIN {X 0,Y 214.364,Z 416.619,A -85,B 0,C 180,E1 -21755.804,E2 -21755.804} C_VEL
LIN {X 0,Y 209.411,Z 419.413,A -85,B 0,C 180,E1 -21758.333,E2 -21758.333} C_VEL
LIN {X 0,Y 206.415,Z 420.459,A -85,B 0,C 180,E1 -21760.091,E2 -21760.091} C_VEL
LIN {X 0,Y 203.653,Z 420.888,A -85,B 0,C 180,E1 -21761.903,E2 -21761.903} C_VEL
LIN {X 0,Y 201.079,Z 420.721,A -85,B 0,C 180,E1 -21763.76,E2 -21763.76} C_VEL
LIN {X 0,Y 198.715,Z 419.946,A -85,B 0,C 180,E1 -21765.664,E2 -21765.664} C_VEL
LIN {X 0,Y 195.759,Z 417.582,A -85,B 0,C 180,E1 -21768.609,E2 -21768.609} C_VEL
LIN {X 0,Y 193.468,Z 413.865,A -85,B 0,C 180,E1 -21771.642,E2 -21771.642} C_VEL
LIN {X 0,Y 192.027,Z 408.527,A -85,B 0,C 180,E1 -21774.748,E2 -21774.748} C_VEL
LIN {X 0,Y 191.43,Z 402.696,A -85,B 0,C 180,E1 -21777.367,E2 -21777.367} C_VEL
LIN {X 0,Y 191.313,Z 395.366,A -85,B 0,C 180,E1 -21779.997,E2 -21779.997} C_VEL
LIN {X 0,Y 191.676,Z 385.842,A -85,B 0,C 180,E1 -21782.624,E2 -21782.624} C_VEL
LIN {X 0,Y 192.136,Z 377.259,A -85,B 0,C 180,E1 -21784.455,E2 -21784.455} C_VEL
LIN {X 0,Y 192.345,Z 367.764,A -85,B 0,C 180,E1 -21786.027,E2 -21786.027} C_VEL
LIN {X 0,Y 192.636,Z 357.914,A -85,B 0,C 180,E1 -21787.268,E2 -21787.268} C_VEL
LIN {X 0,Y 191.68,Z 343.035,A -85,B 0,C 180,E1 -21795.958,E2 -21795.958} C_VEL
LIN {X 0,Y 191.894,Z 335.634,A -85,B 0,C 180,E1 -21800.358,E2 -21800.358} C_VEL
LIN {X 0,Y 192.239,Z 328.107,A -85,B 0,C 180,E1 -21804.857,E2 -21804.857} C_VEL
LIN {X 0,Y 192.667,Z 320.487,A -85,B 0,C 180,E1 -21809.428,E2 -21809.428} C_VEL
LIN {X 0,Y 192.894,Z 320.456,A -85,B 0,C 180,E1 -21810.666,E2 -21810.666} C_VEL
LIN {X 0,Y 192.575,Z 320.495,A -85,B 0,C 180,E1 -21816.593,E2 -21816.593} C_VEL
LIN {X 0,Y 192.501,Z 320.505,A -85,B 0,C 180,E1 -21821.08,E2 -21821.08} C_VEL
LIN {X 0,Y 192.482,Z 320.507,A -85,B 0,C 180,E1 -21826.073,E2 -21826.073} C_VEL
LIN {X 0,Y 192.51,Z 320.502,A -85,B 0,C 180,E1 -21830.049,E2 -21830.049} C_VEL
LIN {X 0,Y 192.552,Z 320.498,A -85,B 0,C 180,E1 -21834.268,E2 -21834.268} C_VEL
LIN {X 0,Y 192.602,Z 320.493,A -85,B 0,C 180,E1 -21837.056,E2 -21837.056} C_VEL
LIN {X 0,Y 192.656,Z 320.484,A -85,B 0,C 180,E1 -21841.69,E2 -21841.69} C_VEL
LIN {X 0,Y 192.697,Z 320.482,A -85,B 0,C 180,E1 -21846.347,E2 -21846.347} C_VEL
LIN {X 0,Y 192.772,Z 320.47,A -85,B 0,C 180,E1 -21851.413,E2 -21851.413} C_VEL
LIN {X 0,Y 192.751,Z 320.472,A -85,B 0,C 180,E1 -21855.213,E2 -21855.213} C_VEL
LIN {X 0,Y 192.935,Z 320.45,A -85,B 0,C 180,E1 -21859.566,E2 -21859.566} C_VEL
LIN {X 0,Y 192.957,Z 320.448,A -85,B 0,C 180,E1 -21863.727,E2 -21863.727} C_VEL
LIN {X 0,Y 193.22,Z 320.415,A -85,B 0,C 180,E1 -21867.916,E2 -21867.916} C_VEL
LIN {X 0,Y 193.403,Z 320.396,A -85,B 0,C 180,E1 -21870,E2 -21870} C_VEL
LIN {X 0,Y 192.929,Z 320.449,A -85,B 0,C 180,E1 -21874.178,E2 -21874.178} C_VEL
LIN {X 0,Y 193.016,Z 320.441,A -85,B 0,C 180,E1 -21878.375,E2 -21878.375} C_VEL
LIN {X 0,Y 192.789,Z 320.464,A -85,B 0,C 180,E1 -21882.634,E2 -21882.634} C_VEL
LIN {X 0,Y 192.76,Z 320.473,A -85,B 0,C 180,E1 -21886.959,E2 -21886.959} C_VEL
LIN {X 0,Y 192.658,Z 320.483,A -85,B 0,C 180,E1 -21891.395,E2 -21891.395} C_VEL
LIN {X 0,Y 192.66,Z 320.485,A -85,B 0,C 180,E1 -21894.229,E2 -21894.229} C_VEL
LIN {X 0,Y 192.641,Z 320.486,A -85,B 0,C 180,E1 -21898.894,E2 -21898.894} C_VEL
LIN {X 0,Y 192.591,Z 320.496,A -85,B 0,C 180,E1 -21903.188,E2 -21903.188} C_VEL
LIN {X 0,Y 192.543,Z 320.496,A -85,B 0,C 180,E1 -21908.354,E2 -21908.354} C_VEL
LIN {X 0,Y 192.482,Z 320.51,A -85,B 0,C 180,E1 -21913.097,E2 -21913.097} C_VEL
LIN {X 0,Y 192.48,Z 320.506,A -85,B 0,C 180,E1 -21916.908,E2 -21916.908} C_VEL
LIN {X 0,Y 192.554,Z 320.498,A -85,B 0,C 180,E1 -21921.653,E2 -21921.653} C_VEL
LIN {X 0,Y 192.886,Z 320.457,A -85,B 0,C 180,E1 -21926.933,E2 -21926.933} C_VEL
LIN {X 0,Y 193.023,Z 320.598,A -85,B 0,C 180,E1 -21928.596,E2 -21928.596} C_VEL
LIN {X 0,Y 192.374,Z 325.214,A -85,B 0,C 180,E1 -21932.831,E2 -21932.831} C_VEL
LIN {X 0,Y 191.819,Z 330.256,A -85,B 0,C 180,E1 -21937.378,E2 -21937.378} C_VEL
LIN {X 0,Y 191.227,Z 336.501,A -85,B 0,C 180,E1 -21942.904,E2 -21942.904} C_VEL
LIN {X 0,Y 191.122,Z 342.422,A -85,B 0,C 180,E1 -21948.065,E2 -21948.065} C_VEL
LIN {X 0,Y 192.542,Z 356.994,A -85,B 0,C 180,E1 -21949.873,E2 -21949.873} C_VEL
LIN {X 0,Y 192.324,Z 366.27,A -85,B 0,C 180,E1 -21951.393,E2 -21951.393} C_VEL
LIN {X 0,Y 191.807,Z 377.552,A -85,B 0,C 180,E1 -21953.692,E2 -21953.692} C_VEL
LIN {X 0,Y 191.504,Z 385.897,A -85,B 0,C 180,E1 -21955.794,E2 -21955.794} C_VEL
LIN {X 0,Y 191.114,Z 394.318,A -85,B 0,C 180,E1 -21958.422,E2 -21958.422} C_VEL
LIN {X 0,Y 191.146,Z 401.303,A -85,B 0,C 180,E1 -21961.056,E2 -21961.056} C_VEL
LIN {X 0,Y 191.667,Z 408.062,A -85,B 0,C 180,E1 -21964.208,E2 -21964.208} C_VEL
LIN {X 0,Y 192.899,Z 413.256,A -85,B 0,C 180,E1 -21967.329,E2 -21967.329} C_VEL
LIN {X 0,Y 194.84,Z 417.208,A -85,B 0,C 180,E1 -21970.393,E2 -21970.393} C_VEL
LIN {X 0,Y 196.535,Z 419.149,A -85,B 0,C 180,E1 -21972.392,E2 -21972.392} C_VEL
LIN {X 0,Y 198.568,Z 420.556,A -85,B 0,C 180,E1 -21974.347,E2 -21974.347} C_VEL
LIN {X 0,Y 200.877,Z 421.489,A -85,B 0,C 180,E1 -21976.256,E2 -21976.256} C_VEL
LIN {X 0,Y 203.455,Z 421.876,A -85,B 0,C 180,E1 -21978.115,E2 -21978.115} C_VEL
LIN {X 0,Y 206.288,Z 421.806,A -85,B 0,C 180,E1 -21979.921,E2 -21979.921} C_VEL
LIN {X 0,Y 209.366,Z 421.233,A -85,B 0,C 180,E1 -21981.672,E2 -21981.672} C_VEL
LIN {X 0,Y 212.609,Z 420.188,A -85,B 0,C 180,E1 -21983.373,E2 -21983.373} C_VEL
LIN {X 0,Y 218.035,Z 417.705,A -85,B 0,C 180,E1 -21985.797,E2 -21985.797} C_VEL
LIN {X 0,Y 220.535,Z 416.263,A -85,B 0,C 180,E1 -21986.835,E2 -21986.835} C_VEL
LIN {X 0,Y 223.011,Z 414.463,A -85,B 0,C 180,E1 -21988.213,E2 -21988.213} C_VEL
LIN {X 0,Y 224.874,Z 412.64,A -85,B 0,C 180,E1 -21990.005,E2 -21990.005} C_VEL
LIN {X 0,Y 226.564,Z 410.745,A -85,B 0,C 180,E1 -21991.828,E2 -21991.828} C_VEL
LIN {X 0,Y 228.041,Z 409.052,A -85,B 0,C 180,E1 -21993.695,E2 -21993.695} C_VEL
LIN {X 0,Y 229.211,Z 407.596,A -85,B 0,C 180,E1 -21995.634,E2 -21995.634} C_VEL
LIN {X 0,Y 229.762,Z 406.869,A -85,B 0,C 180,E1 -21997.72,E2 -21997.72} C_VEL
LIN {X 0,Y 230.286,Z 406.667,A -85,B 0,C 180,E1 -22000.273,E2 -22000.273} C_VEL
LIN {X 0,Y 230.877,Z 407.24,A -85,B 0,C 180,E1 -22003.065,E2 -22003.065} C_VEL
LIN {X 0,Y 231.457,Z 409.518,A -85,B 0,C 180,E1 -22006.783,E2 -22006.783} C_VEL
LIN {X 0,Y 231.641,Z 410.754,A -85,B 0,C 180,E1 -22008.127,E2 -22008.127} C_VEL
LIN {X 0,Y 231.586,Z 412.229,A -85,B 0,C 180,E1 -22009.351,E2 -22009.351} C_VEL
LIN {X 0,Y 230.711,Z 414.029,A -85,B 0,C 180,E1 -22010.23,E2 -22010.23} C_VEL
LIN {X 0,Y 226.322,Z 420.322,A -85,B 0,C 180,E1 -22012.732,E2 -22012.732} C_VEL
LIN {X 0,Y 222.895,Z 424.404,A -85,B 0,C 180,E1 -22014.316,E2 -22014.316} C_VEL
LIN {X 0,Y 214.964,Z 431.766,A -85,B 0,C 180,E1 -22017.354,E2 -22017.354} C_VEL
LIN {X 0,Y 209.619,Z 436.176,A -85,B 0,C 180,E1 -22019.807,E2 -22019.807} C_VEL
LIN {X 0,Y 203.352,Z 440.702,A -85,B 0,C 180,E1 -22023.302,E2 -22023.302} C_VEL
LIN {X 0,Y 198.415,Z 443.861,A -85,B 0,C 180,E1 -22027.069,E2 -22027.069} C_VEL
LIN {X 0,Y 194.753,Z 445.662,A -85,B 0,C 180,E1 -22031.048,E2 -22031.048} C_VEL
LIN {X 0,Y 192.433,Z 446.211,A -85,B 0,C 180,E1 -22035.188,E2 -22035.188} C_VEL
LIN {X 0,Y 191.478,Z 445.446,A -85,B 0,C 180,E1 -22039.425,E2 -22039.425} C_VEL
LIN {X 0,Y 191.735,Z 443.346,A -85,B 0,C 180,E1 -22043.687,E2 -22043.687} C_VEL
LIN {X 0,Y 192.549,Z 440.754,A -85,B 0,C 180,E1 -22046.861,E2 -22046.861} C_VEL
LIN {X 0,Y 193.484,Z 437.083,A -85,B 0,C 180,E1 -22050,E2 -22050} C_VEL
LIN {X 0,Y 193.56,Z 436.466,A -85,B 0,C 180,E1 -22050.415,E2 -22050.415} C_VEL
LIN {X 0,Y 193.304,Z 435.524,A -85,B 0,C 180,E1 -22051.495,E2 -22051.495} C_VEL
LIN {X 0,Y 192.399,Z 435.498,A -85,B 0,C 180,E1 -22052.601,E2 -22052.601} C_VEL
LIN {X 0,Y 191.089,Z 436.068,A -85,B 0,C 180,E1 -22053.711,E2 -22053.711} C_VEL
LIN {X 0,Y 186.585,Z 438.835,A -85,B 0,C 180,E1 -22057.094,E2 -22057.094} C_VEL
LIN {X 0,Y 185.217,Z 440.242,A -85,B 0,C 180,E1 -22058.907,E2 -22058.907} C_VEL
LIN {X 0,Y 185.076,Z 440.693,A -85,B 0,C 180,E1 -22059.528,E2 -22059.528} C_VEL
LIN {X 0,Y 185.352,Z 443.003,A -85,B 0,C 180,E1 -22063.15,E2 -22063.15} C_VEL
LIN {X 0,Y 186.123,Z 443.736,A -85,B 0,C 180,E1 -22065.327,E2 -22065.327} C_VEL
LIN {X 0,Y 187.261,Z 443.977,A -85,B 0,C 180,E1 -22067.472,E2 -22067.472} C_VEL
LIN {X 0,Y 188.952,Z 443.755,A -85,B 0,C 180,E1 -22069.558,E2 -22069.558} C_VEL
LIN {X 0,Y 190.96,Z 443.024,A -85,B 0,C 180,E1 -22071.595,E2 -22071.595} C_VEL
LIN {X 0,Y 193.356,Z 441.807,A -85,B 0,C 180,E1 -22073.567,E2 -22073.567} C_VEL
LIN {X 0,Y 197.663,Z 439.073,A -85,B 0,C 180,E1 -22076.388,E2 -22076.388} C_VEL
LIN {X 0,Y 202.758,Z 434.988,A -85,B 0,C 180,E1 -22079.03,E2 -22079.03} C_VEL
LIN {X 0,Y 208.558,Z 429.572,A -85,B 0,C 180,E1 -22081.488,E2 -22081.488} C_VEL
LIN {X 0,Y 213.921,Z 423.648,A -85,B 0,C 180,E1 -22083.387,E2 -22083.387} C_VEL
LIN {X 0,Y 219.52,Z 415.529,A -85,B 0,C 180,E1 -22085.753,E2 -22085.753} C_VEL
LIN {X 0,Y 222.989,Z 407.757,A -85,B 0,C 180,E1 -22088.353,E2 -22088.353} C_VEL
LIN {X 0,Y 224.451,Z 403.796,A -85,B 0,C 180,E1 -22089.803,E2 -22089.803} C_VEL
LIN {X 0,Y 224.275,Z 402.152,A -85,B 0,C 180,E1 -22091.227,E2 -22091.227} C_VEL
LIN {X 0,Y 223.668,Z 400.469,A -85,B 0,C 180,E1 -22093.731,E2 -22093.731} C_VEL
LIN {X 0,Y 222.944,Z 399.962,A -85,B 0,C 180,E1 -22096.473,E2 -22096.473} C_VEL
LIN {X 0,Y 222.265,Z 400.558,A -85,B 0,C 180,E1 -22099.366,E2 -22099.366} C_VEL
LIN {X 0,Y 221.601,Z 402.375,A -85,B 0,C 180,E1 -22102.454,E2 -22102.454} C_VEL
LIN {X 0,Y 221.196,Z 403.543,A -85,B 0,C 180,E1 -22103.878,E2 -22103.878} C_VEL
LIN {X 0,Y 219.091,Z 407.582,A -85,B 0,C 180,E1 -22106.951,E2 -22106.951} C_VEL
LIN {X 0,Y 216.73,Z 411.503,A -85,B 0,C 180,E1 -22109.824,E2 -22109.824} C_VEL
LIN {X 0,Y 214.925,Z 413.901,A -85,B 0,C 180,E1 -22111.694,E2 -22111.694} C_VEL
LIN {X 0,Y 213.68,Z 415.111,A -85,B 0,C 180,E1 -22112.58,E2 -22112.58} C_VEL
LIN {X 0,Y 209.944,Z 417.715,A -85,B 0,C 180,E1 -22114.201,E2 -22114.201} C_VEL
LIN {X 0,Y 206.368,Z 419.669,A -85,B 0,C 180,E1 -22115.876,E2 -22115.876} C_VEL
LIN {X 0,Y 202.983,Z 420.997,A -85,B 0,C 180,E1 -22117.611,E2 -22117.611} C_VEL
LIN {X 0,Y 199.835,Z 421.698,A -85,B 0,C 180,E1 -22119.407,E2 -22119.407} C_VEL
LIN {X 0,Y 196.956,Z 421.797,A -85,B 0,C 180,E1 -22121.265,E2 -22121.265} C_VEL
LIN {X 0,Y 194.282,Z 421.309,A -85,B 0,C 180,E1 -22123.176,E2 -22123.176} C_VEL
LIN {X 0,Y 191.86,Z 420.215,A -85,B 0,C 180,E1 -22125.14,E2 -22125.14} C_VEL
LIN {X 0,Y 188.818,Z 417.469,A -85,B 0,C 180,E1 -22128.184,E2 -22128.184} C_VEL
LIN {X 0,Y 186.482,Z 413.187,A -85,B 0,C 180,E1 -22131.327,E2 -22131.327} C_VEL
LIN {X 0,Y 185.052,Z 407.36,A -85,B 0,C 180,E1 -22134.549,E2 -22134.549} C_VEL
LIN {X 0,Y 184.477,Z 401.073,A -85,B 0,C 180,E1 -22137.268,E2 -22137.268} C_VEL
LIN {X 0,Y 184.456,Z 393.064,A -85,B 0,C 180,E1 -22139.997,E2 -22139.997} C_VEL
LIN {X 0,Y 184.814,Z 383.922,A -85,B 0,C 180,E1 -22142.449,E2 -22142.449} C_VEL
LIN {X 0,Y 185.251,Z 374.739,A -85,B 0,C 180,E1 -22144.349,E2 -22144.349} C_VEL
LIN {X 0,Y 185.514,Z 364.081,A -85,B 0,C 180,E1 -22145.977,E2 -22145.977} C_VEL
LIN {X 0,Y 185.66,Z 358.648,A -85,B 0,C 180,E1 -22146.654,E2 -22146.654} C_VEL
LIN {X 0,Y 184.603,Z 342.061,A -85,B 0,C 180,E1 -22156.588,E2 -22156.588} C_VEL
LIN {X 0,Y 184.835,Z 334.535,A -85,B 0,C 180,E1 -22161.172,E2 -22161.172} C_VEL
LIN {X 0,Y 185.246,Z 326.861,A -85,B 0,C 180,E1 -22165.864,E2 -22165.864} C_VEL
LIN {X 0,Y 185.587,Z 321.369,A -85,B 0,C 180,E1 -22169.357,E2 -22169.357} C_VEL
LIN {X 0,Y 185.696,Z 321.351,A -85,B 0,C 180,E1 -22171.992,E2 -22171.992} C_VEL
LIN {X 0,Y 185.494,Z 321.38,A -85,B 0,C 180,E1 -22177.312,E2 -22177.312} C_VEL
LIN {X 0,Y 185.458,Z 321.383,A -85,B 0,C 180,E1 -22180.72,E2 -22180.72} C_VEL
LIN {X 0,Y 185.451,Z 321.383,A -85,B 0,C 180,E1 -22186.053,E2 -22186.053} C_VEL
LIN {X 0,Y 185.46,Z 321.38,A -85,B 0,C 180,E1 -22189.893,E2 -22189.893} C_VEL
LIN {X 0,Y 185.498,Z 321.376,A -85,B 0,C 180,E1 -22192.709,E2 -22192.709} C_VEL
LIN {X 0,Y 185.538,Z 321.371,A -85,B 0,C 180,E1 -22197.974,E2 -22197.974} C_VEL
LIN {X 0,Y 185.574,Z 321.365,A -85,B 0,C 180,E1 -22200.574,E2 -22200.574} C_VEL
LIN {X 0,Y 185.579,Z 321.367,A -85,B 0,C 180,E1 -22205.381,E2 -22205.381} C_VEL
LIN {X 0,Y 185.685,Z 321.354,A -85,B 0,C 180,E1 -22211.115,E2 -22211.115} C_VEL
LIN {X 0,Y 185.686,Z 321.354,A -85,B 0,C 180,E1 -22214.636,E2 -22214.636} C_VEL
LIN {X 0,Y 185.878,Z 321.329,A -85,B 0,C 180,E1 -22219.418,E2 -22219.418} C_VEL
LIN {X 0,Y 185.922,Z 321.324,A -85,B 0,C 180,E1 -22223.488,E2 -22223.488} C_VEL
LIN {X 0,Y 186.166,Z 321.294,A -85,B 0,C 180,E1 -22227.836,E2 -22227.836} C_VEL
LIN {X 0,Y 186.369,Z 321.272,A -85,B 0,C 180,E1 -22230,E2 -22230} C_VEL
LIN {X 0,Y 185.877,Z 321.327,A -85,B 0,C 180,E1 -22234.337,E2 -22234.337} C_VEL
LIN {X 0,Y 185.965,Z 321.319,A -85,B 0,C 180,E1 -22238.695,E2 -22238.695} C_VEL
LIN {X 0,Y 185.717,Z 321.346,A -85,B 0,C 180,E1 -22243.124,E2 -22243.124} C_VEL
LIN {X 0,Y 185.707,Z 321.354,A -85,B 0,C 180,E1 -22247.623,E2 -22247.623} C_VEL
LIN {X 0,Y 185.607,Z 321.361,A -85,B 0,C 180,E1 -22252.25,E2 -22252.25} C_VEL
LIN {X 0,Y 185.555,Z 321.371,A -85,B 0,C 180,E1 -22257.033,E2 -22257.033} C_VEL
LIN {X 0,Y 185.571,Z 321.366,A -85,B 0,C 180,E1 -22259.495,E2 -22259.495} C_VEL
LIN {X 0,Y 185.491,Z 321.379,A -85,B 0,C 180,E1 -22264.634,E2 -22264.634} C_VEL
LIN {X 0,Y 185.498,Z 321.375,A -85,B 0,C 180,E1 -22267.315,E2 -22267.315} C_VEL
LIN {X 0,Y 185.463,Z 321.381,A -85,B 0,C 180,E1 -22270.727,E2 -22270.727} C_VEL
LIN {X 0,Y 185.45,Z 321.38,A -85,B 0,C 180,E1 -22276.058,E2 -22276.058} C_VEL
LIN {X 0,Y 185.458,Z 321.381,A -85,B 0,C 180,E1 -22279.897,E2 -22279.897} C_VEL
LIN {X 0,Y 185.658,Z 321.353,A -85,B 0,C 180,E1 -22285.406,E2 -22285.406} C_VEL
LIN {X 0,Y 185.923,Z 321.423,A -85,B 0,C 180,E1 -22288.688,E2 -22288.688} C_VEL
LIN {X 0,Y 185.267,Z 325.908,A -85,B 0,C 180,E1 -22292.925,E2 -22292.925} C_VEL
LIN {X 0,Y 184.689,Z 330.974,A -85,B 0,C 180,E1 -22297.637,E2 -22297.637} C_VEL
LIN {X 0,Y 184.159,Z 336.365,A -85,B 0,C 180,E1 -22302.567,E2 -22302.567} C_VEL
LIN {X 0,Y 184.108,Z 342.867,A -85,B 0,C 180,E1 -22308.372,E2 -22308.372} C_VEL
LIN {X 0,Y 185.406,Z 356.001,A -85,B 0,C 180,E1 -22310.008,E2 -22310.008} C_VEL
LIN {X 0,Y 185.491,Z 360.948,A -85,B 0,C 180,E1 -22310.771,E2 -22310.771} C_VEL
LIN {X 0,Y 184.963,Z 372.279,A -85,B 0,C 180,E1 -22312.909,E2 -22312.909} C_VEL
LIN {X 0,Y 184.673,Z 382.562,A -85,B 0,C 180,E1 -22315.364,E2 -22315.364} C_VEL
LIN {X 0,Y 184.168,Z 392.536,A -85,B 0,C 180,E1 -22318.363,E2 -22318.363} C_VEL
LIN {X 0,Y 184.202,Z 401.262,A -85,B 0,C 180,E1 -22321.643,E2 -22321.643} C_VEL
LIN {X 0,Y 184.817,Z 408.086,A -85,B 0,C 180,E1 -22324.911,E2 -22324.911} C_VEL
LIN {X 0,Y 185.871,Z 412.706,A -85,B 0,C 180,E1 -22327.608,E2 -22327.608} C_VEL
LIN {X 0,Y 187.859,Z 416.999,A -85,B 0,C 180,E1 -22330.784,E2 -22330.784} C_VEL
LIN {X 0,Y 189.629,Z 419.205,A -85,B 0,C 180,E1 -22332.851,E2 -22332.851} C_VEL
LIN {X 0,Y 191.723,Z 420.87,A -85,B 0,C 180,E1 -22334.871,E2 -22334.871} C_VEL
LIN {X 0,Y 194.083,Z 422.052,A -85,B 0,C 180,E1 -22336.842,E2 -22336.842} C_VEL
LIN {X 0,Y 196.774,Z 422.723,A -85,B 0,C 180,E1 -22338.753,E2 -22338.753} C_VEL
LIN {X 0,Y 199.699,Z 422.905,A -85,B 0,C 180,E1 -22340.608,E2 -22340.608} C_VEL
LIN {X 0,Y 202.877,Z 422.619,A -85,B 0,C 180,E1 -22342.402,E2 -22342.402} C_VEL
LIN {X 0,Y 206.275,Z 421.861,A -85,B 0,C 180,E1 -22344.135,E2 -22344.135} C_VEL
LIN {X 0,Y 209.943,Z 420.645,A -85,B 0,C 180,E1 -22345.8,E2 -22345.8} C_VEL
LIN {X 0,Y 213.791,Z 418.9,A -85,B 0,C 180,E1 -22347.404,E2 -22347.404} C_VEL
LIN {X 0,Y 217.25,Z 416.969,A -85,B 0,C 180,E1 -22349.138,E2 -22349.138} C_VEL
LIN {X 0,Y 219.172,Z 415.463,A -85,B 0,C 180,E1 -22350.87,E2 -22350.87} C_VEL
LIN {X 0,Y 221.018,Z 413.918,A -85,B 0,C 180,E1 -22352.725,E2 -22352.725} C_VEL
LIN {X 0,Y 222.745,Z 412.333,A -85,B 0,C 180,E1 -22354.88,E2 -22354.88} C_VEL
LIN {X 0,Y 223.758,Z 411.488,A -85,B 0,C 180,E1 -22356.641,E2 -22356.641} C_VEL
LIN {X 0,Y 224.364,Z 411.118,A -85,B 0,C 180,E1 -22358.794,E2 -22358.794} C_VEL
LIN {X 0,Y 224.938,Z 411.283,A -85,B 0,C 180,E1 -22361.422,E2 -22361.422} C_VEL
LIN {X 0,Y 225.48,Z 412.24,A -85,B 0,C 180,E1 -22364.202,E2 -22364.202} C_VEL
LIN {X 0,Y 225.848,Z 413.939,A -85,B 0,C 180,E1 -22366.795,E2 -22366.795} C_VEL
LIN {X 0,Y 225.894,Z 415.347,A -85,B 0,C 180,E1 -22368.307,E2 -22368.307} C_VEL
LIN {X 0,Y 225.485,Z 416.497,A -85,B 0,C 180,E1 -22369.115,E2 -22369.115} C_VEL
LIN {X 0,Y 222.545,Z 420.309,A -85,B 0,C 180,E1 -22370.831,E2 -22370.831} C_VEL
LIN {X 0,Y 219.211,Z 424.083,A -85,B 0,C 180,E1 -22372.472,E2 -22372.472} C_VEL
LIN {X 0,Y 213.16,Z 429.503,A -85,B 0,C 180,E1 -22374.761,E2 -22374.761} C_VEL
LIN {X 0,Y 207.131,Z 434.102,A -85,B 0,C 180,E1 -22377.12,E2 -22377.12} C_VEL
LIN {X 0,Y 200.128,Z 438.886,A -85,B 0,C 180,E1 -22380.551,E2 -22380.551} C_VEL
LIN {X 0,Y 194.33,Z 442.237,A -85,B 0,C 180,E1 -22384.279,E2 -22384.279} C_VEL
LIN {X 0,Y 189.842,Z 444.321,A -85,B 0,C 180,E1 -22388.272,E2 -22388.272} C_VEL
LIN {X 0,Y 186.665,Z 445.092,A -85,B 0,C 180,E1 -22392.47,E2 -22392.47} C_VEL
LIN {X 0,Y 184.922,Z 444.646,A -85,B 0,C 180,E1 -22396.819,E2 -22396.819} C_VEL
LIN {X 0,Y 184.571,Z 442.909,A -85,B 0,C 180,E1 -22401.239,E2 -22401.239} C_VEL
LIN {X 0,Y 185.441,Z 439.767,A -85,B 0,C 180,E1 -22405.653,E2 -22405.653} C_VEL
LIN {X 0,Y 186.153,Z 437.585,A -85,B 0,C 180,E1 -22407.836,E2 -22407.836} C_VEL
LIN {X 0,Y 187.004,Z 433.164,A -85,B 0,C 180,E1 -22411.077,E2 -22411.077} C_VEL
LIN {X 0,Y 187.506,Z 431.451,A -85,B 0,C 180,E1 -22412.282,E2 -22412.282} C_VEL
LIN {X 0,Y 185.996,Z 436.393,A -85,B 0,C 180,E1 -22415.421,E2 -22415.421} C_VEL
LIN {X 0,Y 185.138,Z 440.052,A -85,B 0,C 180,E1 -22418.734,E2 -22418.734} C_VEL
LIN {X 0,Y 185.076,Z 440.693,A -85,B 0,C 180,E1 -22419.528,E2 -22419.528} C_VEL
LIN {X 0,Y 184.431,Z 441.818,A -85,B 0,C 180,E1 -22421.321,E2 -22421.321} C_VEL
LIN {X 0,Y 182.209,Z 442.614,A -85,B 0,C 180,E1 -22424.337,E2 -22424.337} C_VEL
LIN {X 0,Y 180.816,Z 442.833,A -85,B 0,C 180,E1 -22427.429,E2 -22427.429} C_VEL
LIN {X 0,Y 181.458,Z 442.823,A -85,B 0,C 180,E1 -22429.28,E2 -22429.28} C_VEL
LIN {X 0,Y 184.396,Z 442.471,A -85,B 0,C 180,E1 -22432.404,E2 -22432.404} C_VEL
LIN {X 0,Y 186.877,Z 441.591,A -85,B 0,C 180,E1 -22434.437,E2 -22434.437} C_VEL
LIN {X 0,Y 189.737,Z 440.212,A -85,B 0,C 180,E1 -22436.391,E2 -22436.391} C_VEL
LIN {X 0,Y 194.78,Z 437.126,A -85,B 0,C 180,E1 -22439.151,E2 -22439.151} C_VEL
LIN {X 0,Y 200.496,Z 432.851,A -85,B 0,C 180,E1 -22441.722,E2 -22441.722} C_VEL
LIN {X 0,Y 207.027,Z 427.006,A -85,B 0,C 180,E1 -22444.065,E2 -22444.065} C_VEL
LIN {X 0,Y 210.273,Z 423.57,A -85,B 0,C 180,E1 -22445.208,E2 -22445.208} C_VEL
LIN {X 0,Y 214.575,Z 418.053,A -85,B 0,C 180,E1 -22446.92,E2 -22446.92} C_VEL
LIN {X 0,Y 218.4,Z 411.207,A -85,B 0,C 180,E1 -22449.435,E2 -22449.435} C_VEL
LIN {X 0,Y 219.712,Z 408.661,A -85,B 0,C 180,E1 -22450.429,E2 -22450.429} C_VEL
LIN {X 0,Y 219.455,Z 406.953,A -85,B 0,C 180,E1 -22452.262,E2 -22452.262} C_VEL
LIN {X 0,Y 218.795,Z 405.683,A -85,B 0,C 180,E1 -22455.033,E2 -22455.033} C_VEL
LIN {X 0,Y 218.042,Z 405.592,A -85,B 0,C 180,E1 -22457.846,E2 -22457.846} C_VEL
LIN {X 0,Y 217.031,Z 406.684,A -85,B 0,C 180,E1 -22461.003,E2 -22461.003} C_VEL
LIN {X 0,Y 216.72,Z 407.225,A -85,B 0,C 180,E1 -22461.962,E2 -22461.962} C_VEL
LIN {X 0,Y 215.629,Z 408.946,A -85,B 0,C 180,E1 -22464.076,E2 -22464.076} C_VEL
LIN {X 0,Y 213.083,Z 412.36,A -85,B 0,C 180,E1 -22467.027,E2 -22467.027} C_VEL
LIN {X 0,Y 210.197,Z 415.649,A -85,B 0,C 180,E1 -22469.896,E2 -22469.896} C_VEL
LIN {X 0,Y 208.962,Z 416.761,A -85,B 0,C 180,E1 -22470.981,E2 -22470.981} C_VEL
LIN {X 0,Y 206.548,Z 418.42,A -85,B 0,C 180,E1 -22472.212,E2 -22472.212} C_VEL
LIN {X 0,Y 203.822,Z 419.954,A -85,B 0,C 180,E1 -22473.366,E2 -22473.366} C_VEL
LIN {X 0,Y 200.09,Z 421.527,A -85,B 0,C 180,E1 -22475.069,E2 -22475.069} C_VEL
LIN {X 0,Y 196.569,Z 422.481,A -85,B 0,C 180,E1 -22476.838,E2 -22476.838} C_VEL
LIN {X 0,Y 193.281,Z 422.852,A -85,B 0,C 180,E1 -22478.675,E2 -22478.675} C_VEL
LIN {X 0,Y 190.284,Z 422.621,A -85,B 0,C 180,E1 -22480.582,E2 -22480.582} C_VEL
LIN {X 0,Y 187.501,Z 421.801,A -85,B 0,C 180,E1 -22482.548,E2 -22482.548} C_VEL
LIN {X 0,Y 183.88,Z 419.404,A -85,B 0,C 180,E1 -22485.612,E2 -22485.612} C_VEL
LIN {X 0,Y 180.962,Z 415.674,A -85,B 0,C 180,E1 -22488.8,E2 -22488.8} C_VEL
LIN {X 0,Y 178.94,Z 410.406,A -85,B 0,C 180,E1 -22492.096,E2 -22492.096} C_VEL
LIN {X 0,Y 177.948,Z 404.676,A -85,B 0,C 180,E1 -22494.899,E2 -22494.899} C_VEL
LIN {X 0,Y 177.541,Z 397.588,A -85,B 0,C 180,E1 -22497.728,E2 -22497.728} C_VEL
LIN {X 0,Y 177.644,Z 389.418,A -85,B 0,C 180,E1 -22500.28,E2 -22500.28} C_VEL
LIN {X 0,Y 178.108,Z 380.417,A -85,B 0,C 180,E1 -22502.541,E2 -22502.541} C_VEL
LIN {X 0,Y 178.388,Z 373.289,A -85,B 0,C 180,E1 -22503.95,E2 -22503.95} C_VEL
LIN {X 0,Y 178.639,Z 363.188,A -85,B 0,C 180,E1 -22505.5,E2 -22505.5} C_VEL
LIN {X 0,Y 178.74,Z 359.333,A -85,B 0,C 180,E1 -22505.992,E2 -22505.992} C_VEL
LIN {X 0,Y 177.479,Z 342.873,A -85,B 0,C 180,E1 -22516.089,E2 -22516.089} C_VEL
LIN {X 0,Y 177.727,Z 335.256,A -85,B 0,C 180,E1 -22520.845,E2 -22520.845} C_VEL
LIN {X 0,Y 178.132,Z 327.496,A -85,B 0,C 180,E1 -22525.718,E2 -22525.718} C_VEL
LIN {X 0,Y 178.465,Z 322.256,A -85,B 0,C 180,E1 -22529.06,E2 -22529.06} C_VEL
LIN {X 0,Y 178.574,Z 322.24,A -85,B 0,C 180,E1 -22530.769,E2 -22530.769} C_VEL
LIN {X 0,Y 178.518,Z 322.241,A -85,B 0,C 180,E1 -22534.234,E2 -22534.234} C_VEL
LIN {X 0,Y 178.383,Z 322.266,A -85,B 0,C 180,E1 -22539.074,E2 -22539.074} C_VEL
LIN {X 0,Y 178.388,Z 322.259,A -85,B 0,C 180,E1 -22542.043,E2 -22542.043} C_VEL
LIN {X 0,Y 178.386,Z 322.265,A -85,B 0,C 180,E1 -22545.162,E2 -22545.162} C_VEL
LIN {X 0,Y 178.395,Z 322.263,A -85,B 0,C 180,E1 -22548.457,E2 -22548.457} C_VEL
LIN {X 0,Y 178.415,Z 322.258,A -85,B 0,C 180,E1 -22553.781,E2 -22553.781} C_VEL
LIN {X 0,Y 178.479,Z 322.254,A -85,B 0,C 180,E1 -22556.545,E2 -22556.545} C_VEL
LIN {X 0,Y 178.515,Z 322.243,A -85,B 0,C 180,E1 -22560.004,E2 -22560.004} C_VEL
LIN {X 0,Y 178.526,Z 322.247,A -85,B 0,C 180,E1 -22564.874,E2 -22564.874} C_VEL
LIN {X 0,Y 178.629,Z 322.234,A -85,B 0,C 180,E1 -22570.769,E2 -22570.769} C_VEL
LIN {X 0,Y 178.646,Z 322.228,A -85,B 0,C 180,E1 -22576.347,E2 -22576.347} C_VEL
LIN {X 0,Y 178.895,Z 322.2,A -85,B 0,C 180,E1 -22580.959,E2 -22580.959} C_VEL
LIN {X 0,Y 179.114,Z 322.172,A -85,B 0,C 180,E1 -22587.751,E2 -22587.751} C_VEL
LIN {X 0,Y 179.334,Z 322.148,A -85,B 0,C 180,E1 -22590,E2 -22590} C_VEL
LIN {X 0,Y 178.826,Z 322.205,A -85,B 0,C 180,E1 -22594.508,E2 -22594.508} C_VEL
LIN {X 0,Y 178.895,Z 322.2,A -85,B 0,C 180,E1 -22599.041,E2 -22599.041} C_VEL
LIN {X 0,Y 178.646,Z 322.228,A -85,B 0,C 180,E1 -22603.653,E2 -22603.653} C_VEL
LIN {X 0,Y 178.645,Z 322.232,A -85,B 0,C 180,E1 -22609.246,E2 -22609.246} C_VEL
LIN {X 0,Y 178.526,Z 322.247,A -85,B 0,C 180,E1 -22615.126,E2 -22615.126} C_VEL
LIN {X 0,Y 178.471,Z 322.249,A -85,B 0,C 180,E1 -22620.792,E2 -22620.792} C_VEL
LIN {X 0,Y 178.477,Z 322.252,A -85,B 0,C 180,E1 -22624.221,E2 -22624.221} C_VEL
LIN {X 0,Y 178.387,Z 322.26,A -85,B 0,C 180,E1 -22629.077,E2 -22629.077} C_VEL
LIN {X 0,Y 178.39,Z 322.262,A -85,B 0,C 180,E1 -22632.048,E2 -22632.048} C_VEL
LIN {X 0,Y 178.386,Z 322.263,A -85,B 0,C 180,E1 -22635.167,E2 -22635.167} C_VEL
LIN {X 0,Y 178.394,Z 322.259,A -85,B 0,C 180,E1 -22638.463,E2 -22638.463} C_VEL
LIN {X 0,Y 178.514,Z 322.246,A -85,B 0,C 180,E1 -22643.809,E2 -22643.809} C_VEL
LIN {X 0,Y 178.863,Z 322.205,A -85,B 0,C 180,E1 -22648.712,E2 -22648.712} C_VEL
LIN {X 0,Y 178.022,Z 327.867,A -85,B 0,C 180,E1 -22654.265,E2 -22654.265} C_VEL
LIN {X 0,Y 177.43,Z 332.936,A -85,B 0,C 180,E1 -22659.119,E2 -22659.119} C_VEL
LIN {X 0,Y 176.886,Z 339.213,A -85,B 0,C 180,E1 -22665.037,E2 -22665.037} C_VEL
LIN {X 0,Y 177.092,Z 343.203,A -85,B 0,C 180,E1 -22668.682,E2 -22668.682} C_VEL
LIN {X 0,Y 178.3,Z 355.112,A -85,B 0,C 180,E1 -22670.204,E2 -22670.204} C_VEL
LIN {X 0,Y 178.49,Z 359.797,A -85,B 0,C 180,E1 -22670.941,E2 -22670.941} C_VEL
LIN {X 0,Y 178.062,Z 370.21,A -85,B 0,C 180,E1 -22672.918,E2 -22672.918} C_VEL
LIN {X 0,Y 177.732,Z 381.015,A -85,B 0,C 180,E1 -22675.467,E2 -22675.467} C_VEL
LIN {X 0,Y 177.216,Z 390.584,A -85,B 0,C 180,E1 -22678.299,E2 -22678.299} C_VEL
LIN {X 0,Y 177.21,Z 399.714,A -85,B 0,C 180,E1 -22681.707,E2 -22681.707} C_VEL
LIN {X 0,Y 177.804,Z 407.03,A -85,B 0,C 180,E1 -22685.105,E2 -22685.105} C_VEL
LIN {X 0,Y 178.872,Z 411.971,A -85,B 0,C 180,E1 -22687.907,E2 -22687.907} C_VEL
LIN {X 0,Y 180.891,Z 416.63,A -85,B 0,C 180,E1 -22691.204,E2 -22691.204} C_VEL
LIN {X 0,Y 182.72,Z 419.102,A -85,B 0,C 180,E1 -22693.346,E2 -22693.346} C_VEL
LIN {X 0,Y 184.869,Z 421.034,A -85,B 0,C 180,E1 -22695.436,E2 -22695.436} C_VEL
LIN {X 0,Y 187.3,Z 422.459,A -85,B 0,C 180,E1 -22697.471,E2 -22697.471} C_VEL
LIN {X 0,Y 190.094,Z 423.422,A -85,B 0,C 180,E1 -22699.438,E2 -22699.438} C_VEL
LIN {X 0,Y 193.119,Z 423.865,A -85,B 0,C 180,E1 -22701.344,E2 -22701.344} C_VEL
LIN {X 0,Y 196.414,Z 423.876,A -85,B 0,C 180,E1 -22703.181,E2 -22703.181} C_VEL
LIN {X 0,Y 199.926,Z 423.389,A -85,B 0,C 180,E1 -22704.953,E2 -22704.953} C_VEL
LIN {X 0,Y 206.658,Z 421.473,A -85,B 0,C 180,E1 -22707.846,E2 -22707.846} C_VEL
LIN {X 0,Y 211.286,Z 419.457,A -85,B 0,C 180,E1 -22709.933,E2 -22709.933} C_VEL
LIN {X 0,Y 213.458,Z 418.165,A -85,B 0,C 180,E1 -22711.792,E2 -22711.792} C_VEL
LIN {X 0,Y 215.422,Z 416.906,A -85,B 0,C 180,E1 -22713.687,E2 -22713.687} C_VEL
LIN {X 0,Y 217.329,Z 415.675,A -85,B 0,C 180,E1 -22716.055,E2 -22716.055} C_VEL
LIN {X 0,Y 218.128,Z 415.231,A -85,B 0,C 180,E1 -22717.749,E2 -22717.749} C_VEL
LIN {X 0,Y 218.774,Z 415.212,A -85,B 0,C 180,E1 -22719.98,E2 -22719.98} C_VEL
LIN {X 0,Y 219.394,Z 415.735,A -85,B 0,C 180,E1 -22722.542,E2 -22722.542} C_VEL
LIN {X 0,Y 219.811,Z 417.043,A -85,B 0,C 180,E1 -22725.299,E2 -22725.299} C_VEL
LIN {X 0,Y 219.948,Z 418.92,A -85,B 0,C 180,E1 -22727.855,E2 -22727.855} C_VEL
LIN {X 0,Y 218.88,Z 420.465,A -85,B 0,C 180,E1 -22728.835,E2 -22728.835} C_VEL
LIN {X 0,Y 213.762,Z 425.675,A -85,B 0,C 180,E1 -22731.341,E2 -22731.341} C_VEL
LIN {X 0,Y 207.453,Z 430.616,A -85,B 0,C 180,E1 -22733.64,E2 -22733.64} C_VEL
LIN {X 0,Y 199.313,Z 435.981,A -85,B 0,C 180,E1 -22736.869,E2 -22736.869} C_VEL
LIN {X 0,Y 193.986,Z 439.032,A -85,B 0,C 180,E1 -22739.522,E2 -22739.522} C_VEL
LIN {X 0,Y 187.953,Z 441.914,A -85,B 0,C 180,E1 -22743.339,E2 -22743.339} C_VEL
LIN {X 0,Y 183.272,Z 443.571,A -85,B 0,C 180,E1 -22747.451,E2 -22747.451} C_VEL
LIN {X 0,Y 179.933,Z 443.977,A -85,B 0,C 180,E1 -22751.792,E2 -22751.792} C_VEL
LIN {X 0,Y 178.125,Z 443.169,A -85,B 0,C 180,E1 -22756.306,E2 -22756.306} C_VEL
LIN {X 0,Y 177.766,Z 440.902,A -85,B 0,C 180,E1 -22761.271,E2 -22761.271} C_VEL
LIN {X 0,Y 178.662,Z 437.66,A -85,B 0,C 180,E1 -22765.488,E2 -22765.488} C_VEL
LIN {X 0,Y 179.429,Z 435.302,A -85,B 0,C 180,E1 -22767.755,E2 -22767.755} C_VEL
LIN {X 0,Y 180.373,Z 430.64,A -85,B 0,C 180,E1 -22771.116,E2 -22771.116} C_VEL
LIN {X 0,Y 181.019,Z 428.61,A -85,B 0,C 180,E1 -22772.434,E2 -22772.434} C_VEL
LIN {X 0,Y 179.385,Z 433.862,A -85,B 0,C 180,E1 -22775.621,E2 -22775.621} C_VEL
LIN {X 0,Y 178.459,Z 437.877,A -85,B 0,C 180,E1 -22779.063,E2 -22779.063} C_VEL
LIN {X 0,Y 178.29,Z 439.847,A -85,B 0,C 180,E1 -22781.367,E2 -22781.367} C_VEL
LIN {X 0,Y 178.616,Z 441.283,A -85,B 0,C 180,E1 -22783.655,E2 -22783.655} C_VEL
LIN {X 0,Y 179.39,Z 442.264,A -85,B 0,C 180,E1 -22785.917,E2 -22785.917} C_VEL
LIN {X 0,Y 181.458,Z 442.823,A -85,B 0,C 180,E1 -22789.28,E2 -22789.28} C_VEL
LIN {X 0,Y 182.399,Z 442.699,A -85,B 0,C 180,E1 -22791.116,E2 -22791.116} C_VEL
LIN {X 0,Y 182.81,Z 441.712,A -85,B 0,C 180,E1 -22794.209,E2 -22794.209} C_VEL
LIN {X 0,Y 183.986,Z 440.115,A -85,B 0,C 180,E1 -22797.224,E2 -22797.224} C_VEL
LIN {X 0,Y 186.067,Z 438.859,A -85,B 0,C 180,E1 -22798.881,E2 -22798.881} C_VEL
LIN {X 0,Y 190.528,Z 436.49,A -85,B 0,C 180,E1 -22801.092,E2 -22801.092} C_VEL
LIN {X 0,Y 196.683,Z 432.359,A -85,B 0,C 180,E1 -22803.632,E2 -22803.632} C_VEL
LIN {X 0,Y 203.592,Z 426.781,A -85,B 0,C 180,E1 -22805.933,E2 -22805.933} C_VEL
LIN {X 0,Y 209.894,Z 420.12,A -85,B 0,C 180,E1 -22808.276,E2 -22808.276} C_VEL
LIN {X 0,Y 214.564,Z 413.193,A -85,B 0,C 180,E1 -22811.115,E2 -22811.115} C_VEL
LIN {X 0,Y 214.143,Z 411.379,A -85,B 0,C 180,E1 -22813.776,E2 -22813.776} C_VEL
LIN {X 0,Y 213.441,Z 410.702,A -85,B 0,C 180,E1 -22816.419,E2 -22816.419} C_VEL
LIN {X 0,Y 212.353,Z 410.992,A -85,B 0,C 180,E1 -22819.571,E2 -22819.571} C_VEL
LIN {X 0,Y 211.805,Z 411.534,A -85,B 0,C 180,E1 -22820.914,E2 -22820.914} C_VEL
LIN {X 0,Y 210.423,Z 412.976,A -85,B 0,C 180,E1 -22823.282,E2 -22823.282} C_VEL
LIN {X 0,Y 208.745,Z 414.692,A -85,B 0,C 180,E1 -22825.083,E2 -22825.083} C_VEL
LIN {X 0,Y 206.697,Z 416.598,A -85,B 0,C 180,E1 -22827.039,E2 -22827.039} C_VEL
LIN {X 0,Y 203.815,Z 418.895,A -85,B 0,C 180,E1 -22829.549,E2 -22829.549} C_VEL
LIN {X 0,Y 201.741,Z 420.123,A -85,B 0,C 180,E1 -22830.807,E2 -22830.807} C_VEL
LIN {X 0,Y 197.674,Z 421.934,A -85,B 0,C 180,E1 -22832.468,E2 -22832.468} C_VEL
LIN {X 0,Y 193.802,Z 423.13,A -85,B 0,C 180,E1 -22834.201,E2 -22834.201} C_VEL
LIN {X 0,Y 190.151,Z 423.739,A -85,B 0,C 180,E1 -22836.008,E2 -22836.008} C_VEL
LIN {X 0,Y 186.721,Z 423.755,A -85,B 0,C 180,E1 -22837.887,E2 -22837.887} C_VEL
LIN {X 0,Y 183.62,Z 423.175,A -85,B 0,C 180,E1 -22839.848,E2 -22839.848} C_VEL
LIN {X 0,Y 180.731,Z 422.016,A -85,B 0,C 180,E1 -22841.872,E2 -22841.872} C_VEL
LIN {X 0,Y 177.012,Z 419.186,A -85,B 0,C 180,E1 -22845.041,E2 -22845.041} C_VEL
LIN {X 0,Y 174.049,Z 414.901,A -85,B 0,C 180,E1 -22848.349,E2 -22848.349} C_VEL
LIN {X 0,Y 171.999,Z 409.068,A -85,B 0,C 180,E1 -22851.775,E2 -22851.775} C_VEL
LIN {X 0,Y 171.047,Z 402.914,A -85,B 0,C 180,E1 -22854.693,E2 -22854.693} C_VEL
LIN {X 0,Y 170.726,Z 395.079,A -85,B 0,C 180,E1 -22857.638,E2 -22857.638} C_VEL
LIN {X 0,Y 170.879,Z 386.311,A -85,B 0,C 180,E1 -22860.292,E2 -22860.292} C_VEL
LIN {X 0,Y 171.405,Z 377.719,A -85,B 0,C 180,E1 -22862.347,E2 -22862.347} C_VEL
LIN {X 0,Y 171.699,Z 367.932,A -85,B 0,C 180,E1 -22864.105,E2 -22864.105} C_VEL
LIN {X 0,Y 171.86,Z 359.963,A -85,B 0,C 180,E1 -22865.276,E2 -22865.276} C_VEL
LIN {X 0,Y 170.412,Z 341.728,A -85,B 0,C 180,E1 -22876.776,E2 -22876.776} C_VEL
LIN {X 0,Y 170.693,Z 333.988,A -85,B 0,C 180,E1 -22881.747,E2 -22881.747} C_VEL
LIN {X 0,Y 171.146,Z 326.067,A -85,B 0,C 180,E1 -22886.85,E2 -22886.85} C_VEL
LIN {X 0,Y 171.326,Z 323.146,A -85,B 0,C 180,E1 -22888.812,E2 -22888.812} C_VEL
LIN {X 0,Y 171.482,Z 323.122,A -85,B 0,C 180,E1 -22892.19,E2 -22892.19} C_VEL
LIN {X 0,Y 171.408,Z 323.129,A -85,B 0,C 180,E1 -22895.027,E2 -22895.027} C_VEL
LIN {X 0,Y 171.338,Z 323.142,A -85,B 0,C 180,E1 -22898.799,E2 -22898.799} C_VEL
LIN {X 0,Y 171.313,Z 323.141,A -85,B 0,C 180,E1 -22904.215,E2 -22904.215} C_VEL
LIN {X 0,Y 171.327,Z 323.143,A -85,B 0,C 180,E1 -22908.979,E2 -22908.979} C_VEL
LIN {X 0,Y 171.379,Z 323.132,A -85,B 0,C 180,E1 -22912.039,E2 -22912.039} C_VEL
LIN {X 0,Y 171.39,Z 323.136,A -85,B 0,C 180,E1 -22915.09,E2 -22915.09} C_VEL
LIN {X 0,Y 171.441,Z 323.125,A -85,B 0,C 180,E1 -22920.533,E2 -22920.533} C_VEL
LIN {X 0,Y 171.45,Z 323.127,A -85,B 0,C 180,E1 -22925.8,E2 -22925.8} C_VEL
LIN {X 0,Y 171.586,Z 323.111,A -85,B 0,C 180,E1 -22930.872,E2 -22930.872} C_VEL
LIN {X 0,Y 171.567,Z 323.111,A -85,B 0,C 180,E1 -22935.772,E2 -22935.772} C_VEL
LIN {X 0,Y 171.833,Z 323.081,A -85,B 0,C 180,E1 -22940.584,E2 -22940.584} C_VEL
LIN {X 0,Y 171.775,Z 323.083,A -85,B 0,C 180,E1 -22945.306,E2 -22945.306} C_VEL
LIN {X 0,Y 172.299,Z 323.024,A -85,B 0,C 180,E1 -22950,E2 -22950} C_VEL
LIN {X 0,Y 171.775,Z 323.083,A -85,B 0,C 180,E1 -22954.694,E2 -22954.694} C_VEL
LIN {X 0,Y 171.833,Z 323.081,A -85,B 0,C 180,E1 -22959.416,E2 -22959.416} C_VEL
LIN {X 0,Y 171.567,Z 323.111,A -85,B 0,C 180,E1 -22964.228,E2 -22964.228} C_VEL
LIN {X 0,Y 171.566,Z 323.112,A -85,B 0,C 180,E1 -22969.592,E2 -22969.592} C_VEL
LIN {X 0,Y 171.461,Z 323.128,A -85,B 0,C 180,E1 -22975.618,E2 -22975.618} C_VEL
LIN {X 0,Y 171.434,Z 323.125,A -85,B 0,C 180,E1 -22980.589,E2 -22980.589} C_VEL
LIN {X 0,Y 171.385,Z 323.137,A -85,B 0,C 180,E1 -22985.037,E2 -22985.037} C_VEL
LIN {X 0,Y 171.35,Z 323.136,A -85,B 0,C 180,E1 -22988.81,E2 -22988.81} C_VEL
LIN {X 0,Y 171.313,Z 323.144,A -85,B 0,C 180,E1 -22994.22,E2 -22994.22} C_VEL
LIN {X 0,Y 171.329,Z 323.142,A -85,B 0,C 180,E1 -22998.984,E2 -22998.984} C_VEL
LIN {X 0,Y 171.408,Z 323.133,A -85,B 0,C 180,E1 -23002.051,E2 -23002.051} C_VEL
LIN {X 0,Y 171.841,Z 323.077,A -85,B 0,C 180,E1 -23007.885,E2 -23007.885} C_VEL
LIN {X 0,Y 171.752,Z 323.196,A -85,B 0,C 180,E1 -23009.085,E2 -23009.085} C_VEL
LIN {X 0,Y 170.856,Z 328.902,A -85,B 0,C 180,E1 -23014.817,E2 -23014.817} C_VEL
LIN {X 0,Y 170.303,Z 333.618,A -85,B 0,C 180,E1 -23019.469,E2 -23019.469} C_VEL
LIN {X 0,Y 169.768,Z 339.905,A -85,B 0,C 180,E1 -23025.621,E2 -23025.621} C_VEL
LIN {X 0,Y 170.109,Z 343.49,A -85,B 0,C 180,E1 -23029.062,E2 -23029.062} C_VEL
LIN {X 0,Y 171.485,Z 356.831,A -85,B 0,C 180,E1 -23030.865,E2 -23030.865} C_VEL
LIN {X 0,Y 171.22,Z 366.572,A -85,B 0,C 180,E1 -23032.633,E2 -23032.633} C_VEL
LIN {X 0,Y 170.799,Z 378.204,A -85,B 0,C 180,E1 -23035.283,E2 -23035.283} C_VEL
LIN {X 0,Y 170.409,Z 386.424,A -85,B 0,C 180,E1 -23037.639,E2 -23037.639} C_VEL
LIN {X 0,Y 170.202,Z 394.986,A -85,B 0,C 180,E1 -23040.595,E2 -23040.595} C_VEL
LIN {X 0,Y 170.564,Z 403.404,A -85,B 0,C 180,E1 -23044.138,E2 -23044.138} C_VEL
LIN {X 0,Y 171.898,Z 411.017,A -85,B 0,C 180,E1 -23048.23,E2 -23048.23} C_VEL
LIN {X 0,Y 173.94,Z 416.124,A -85,B 0,C 180,E1 -23051.658,E2 -23051.658} C_VEL
LIN {X 0,Y 176.901,Z 419.987,A -85,B 0,C 180,E1 -23054.968,E2 -23054.968} C_VEL
LIN {X 0,Y 180.545,Z 422.717,A -85,B 0,C 180,E1 -23058.147,E2 -23058.147} C_VEL
LIN {X 0,Y 183.415,Z 423.951,A -85,B 0,C 180,E1 -23060.176,E2 -23060.176} C_VEL
LIN {X 0,Y 186.556,Z 424.673,A -85,B 0,C 180,E1 -23062.134,E2 -23062.134} C_VEL
LIN {X 0,Y 189.956,Z 424.963,A -85,B 0,C 180,E1 -23064.018,E2 -23064.018} C_VEL
LIN {X 0,Y 193.61,Z 424.759,A -85,B 0,C 180,E1 -23065.826,E2 -23065.826} C_VEL
LIN {X 0,Y 200.115,Z 423.508,A -85,B 0,C 180,E1 -23068.598,E2 -23068.598} C_VEL
LIN {X 0,Y 205.399,Z 421.721,A -85,B 0,C 180,E1 -23070.883,E2 -23070.883} C_VEL
LIN {X 0,Y 207.72,Z 420.722,A -85,B 0,C 180,E1 -23072.778,E2 -23072.778} C_VEL
LIN {X 0,Y 209.761,Z 419.754,A -85,B 0,C 180,E1 -23074.724,E2 -23074.724} C_VEL
LIN {X 0,Y 211.61,Z 418.967,A -85,B 0,C 180,E1 -23077.146,E2 -23077.146} C_VEL
LIN {X 0,Y 212.372,Z 418.865,A -85,B 0,C 180,E1 -23078.962,E2 -23078.962} C_VEL
LIN {X 0,Y 212.994,Z 419.168,A -85,B 0,C 180,E1 -23081.297,E2 -23081.297} C_VEL
LIN {X 0,Y 213.505,Z 419.963,A -85,B 0,C 180,E1 -23083.733,E2 -23083.733} C_VEL
LIN {X 0,Y 213.819,Z 421.883,A -85,B 0,C 180,E1 -23087,E2 -23087} C_VEL
LIN {X 0,Y 213.273,Z 422.813,A -85,B 0,C 180,E1 -23087.824,E2 -23087.824} C_VEL
LIN {X 0,Y 208.39,Z 427.109,A -85,B 0,C 180,E1 -23090.15,E2 -23090.15} C_VEL
LIN {X 0,Y 201.83,Z 431.584,A -85,B 0,C 180,E1 -23092.456,E2 -23092.456} C_VEL
LIN {X 0,Y 193.433,Z 436.375,A -85,B 0,C 180,E1 -23095.725,E2 -23095.725} C_VEL
LIN {X 0,Y 187.919,Z 439.035,A -85,B 0,C 180,E1 -23098.427,E2 -23098.427} C_VEL
LIN {X 0,Y 181.647,Z 441.466,A -85,B 0,C 180,E1 -23102.336,E2 -23102.336} C_VEL
LIN {X 0,Y 176.744,Z 442.684,A -85,B 0,C 180,E1 -23106.569,E2 -23106.569} C_VEL
LIN {X 0,Y 173.255,Z 442.726,A -85,B 0,C 180,E1 -23111.064,E2 -23111.064} C_VEL
LIN {X 0,Y 171.36,Z 441.566,A -85,B 0,C 180,E1 -23115.754,E2 -23115.754} C_VEL
LIN {X 0,Y 170.971,Z 439.149,A -85,B 0,C 180,E1 -23120.607,E2 -23120.607} C_VEL
LIN {X 0,Y 171.93,Z 435.421,A -85,B 0,C 180,E1 -23125.311,E2 -23125.311} C_VEL
LIN {X 0,Y 172.774,Z 432.88,A -85,B 0,C 180,E1 -23127.669,E2 -23127.669} C_VEL
LIN {X 0,Y 173.799,Z 427.914,A -85,B 0,C 180,E1 -23131.159,E2 -23131.159} C_VEL
LIN {X 0,Y 174.594,Z 425.632,A -85,B 0,C 180,E1 -23132.596,E2 -23132.596} C_VEL
LIN {X 0,Y 173.456,Z 429.298,A -85,B 0,C 180,E1 -23134.648,E2 -23134.648} C_VEL
LIN {X 0,Y 172.081,Z 434.198,A -85,B 0,C 180,E1 -23138.218,E2 -23138.218} C_VEL
LIN {X 0,Y 171.616,Z 437.728,A -85,B 0,C 180,E1 -23141.815,E2 -23141.815} C_VEL
LIN {X 0,Y 171.93,Z 439.46,A -85,B 0,C 180,E1 -23144.197,E2 -23144.197} C_VEL
LIN {X 0,Y 172.724,Z 440.694,A -85,B 0,C 180,E1 -23146.548,E2 -23146.548} C_VEL
LIN {X 0,Y 174.697,Z 441.601,A -85,B 0,C 180,E1 -23149.849,E2 -23149.849} C_VEL
LIN {X 0,Y 177.891,Z 441.668,A -85,B 0,C 180,E1 -23153.271,E2 -23153.271} C_VEL
LIN {X 0,Y 180.449,Z 441.094,A -85,B 0,C 180,E1 -23155.367,E2 -23155.367} C_VEL
LIN {X 0,Y 183.423,Z 440.053,A -85,B 0,C 180,E1 -23157.374,E2 -23157.374} C_VEL
LIN {X 0,Y 186.067,Z 438.859,A -85,B 0,C 180,E1 -23158.881,E2 -23158.881} C_VEL
LIN {X 0,Y 188.429,Z 437.505,A -85,B 0,C 180,E1 -23160.49,E2 -23160.49} C_VEL
LIN {X 0,Y 191.248,Z 434.772,A -85,B 0,C 180,E1 -23163.241,E2 -23163.241} C_VEL
LIN {X 0,Y 194.587,Z 431.297,A -85,B 0,C 180,E1 -23165.786,E2 -23165.786} C_VEL
LIN {X 0,Y 197.662,Z 428.775,A -85,B 0,C 180,E1 -23167.041,E2 -23167.041} C_VEL
LIN {X 0,Y 202.471,Z 424.689,A -85,B 0,C 180,E1 -23168.668,E2 -23168.668} C_VEL
LIN {X 0,Y 205.604,Z 421.638,A -85,B 0,C 180,E1 -23169.86,E2 -23169.86} C_VEL
LIN {X 0,Y 208.378,Z 418.24,A -85,B 0,C 180,E1 -23171.393,E2 -23171.393} C_VEL
LIN {X 0,Y 208.996,Z 417.057,A -85,B 0,C 180,E1 -23172.282,E2 -23172.282} C_VEL
LIN {X 0,Y 208.446,Z 415.724,A -85,B 0,C 180,E1 -23175.076,E2 -23175.076} C_VEL
LIN {X 0,Y 207.391,Z 415.391,A -85,B 0,C 180,E1 -23178.205,E2 -23178.205} C_VEL
LIN {X 0,Y 206.711,Z 415.627,A -85,B 0,C 180,E1 -23179.758,E2 -23179.758} C_VEL
LIN {X 0,Y 205.362,Z 416.568,A -85,B 0,C 180,E1 -23181.972,E2 -23181.972} C_VEL
LIN {X 0,Y 203.465,Z 417.943,A -85,B 0,C 180,E1 -23184.038,E2 -23184.038} C_VEL
LIN {X 0,Y 201.197,Z 419.442,A -85,B 0,C 180,E1 -23186.018,E2 -23186.018} C_VEL
LIN {X 0,Y 198.637,Z 420.997,A -85,B 0,C 180,E1 -23188.119,E2 -23188.119} C_VEL
LIN {X 0,Y 195.789,Z 422.335,A -85,B 0,C 180,E1 -23189.829,E2 -23189.829} C_VEL
LIN {X 0,Y 191.543,Z 423.766,A -85,B 0,C 180,E1 -23191.508,E2 -23191.508} C_VEL
LIN {X 0,Y 187.542,Z 424.582,A -85,B 0,C 180,E1 -23193.273,E2 -23193.273} C_VEL
LIN {X 0,Y 183.736,Z 424.823,A -85,B 0,C 180,E1 -23195.115,E2 -23195.115} C_VEL
LIN {X 0,Y 180.201,Z 424.487,A -85,B 0,C 180,E1 -23197.042,E2 -23197.042} C_VEL
LIN {X 0,Y 176.962,Z 423.564,A -85,B 0,C 180,E1 -23199.054,E2 -23199.054} C_VEL
LIN {X 0,Y 172.653,Z 421.093,A -85,B 0,C 180,E1 -23202.221,E2 -23202.221} C_VEL
LIN {X 0,Y 169.1,Z 417.248,A -85,B 0,C 180,E1 -23205.557,E2 -23205.557} C_VEL
LIN {X 0,Y 166.385,Z 411.992,A -85,B 0,C 180,E1 -23209.04,E2 -23209.04} C_VEL
LIN {X 0,Y 164.663,Z 404.941,A -85,B 0,C 180,E1 -23212.64,E2 -23212.64} C_VEL
LIN {X 0,Y 164.053,Z 397.612,A -85,B 0,C 180,E1 -23215.697,E2 -23215.697} C_VEL
LIN {X 0,Y 164.021,Z 389.357,A -85,B 0,C 180,E1 -23218.462,E2 -23218.462} C_VEL
LIN {X 0,Y 164.433,Z 380.076,A -85,B 0,C 180,E1 -23220.915,E2 -23220.915} C_VEL
LIN {X 0,Y 164.833,Z 371.305,A -85,B 0,C 180,E1 -23222.746,E2 -23222.746} C_VEL
LIN {X 0,Y 165.063,Z 360.658,A -85,B 0,C 180,E1 -23224.423,E2 -23224.423} C_VEL
LIN {X 0,Y 163.299,Z 342.43,A -85,B 0,C 180,E1 -23236.241,E2 -23236.241} C_VEL
LIN {X 0,Y 163.498,Z 336.585,A -85,B 0,C 180,E1 -23240.11,E2 -23240.11} C_VEL
LIN {X 0,Y 163.961,Z 327.96,A -85,B 0,C 180,E1 -23245.823,E2 -23245.823} C_VEL
LIN {X 0,Y 164.229,Z 324.031,A -85,B 0,C 180,E1 -23248.6,E2 -23248.6} C_VEL
LIN {X 0,Y 164.447,Z 324.001,A -85,B 0,C 180,E1 -23251.268,E2 -23251.268} C_VEL
LIN {X 0,Y 164.281,Z 324.02,A -85,B 0,C 180,E1 -23256.788,E2 -23256.788} C_VEL
LIN {X 0,Y 164.28,Z 324.02,A -85,B 0,C 180,E1 -23259.915,E2 -23259.915} C_VEL
LIN {X 0,Y 164.273,Z 324.019,A -85,B 0,C 180,E1 -23263.339,E2 -23263.339} C_VEL
LIN {X 0,Y 164.256,Z 324.025,A -85,B 0,C 180,E1 -23266.796,E2 -23266.796} C_VEL
LIN {X 0,Y 164.288,Z 324.018,A -85,B 0,C 180,E1 -23270.35,E2 -23270.35} C_VEL
LIN {X 0,Y 164.322,Z 324.015,A -85,B 0,C 180,E1 -23274.347,E2 -23274.347} C_VEL
LIN {X 0,Y 164.383,Z 324.003,A -85,B 0,C 180,E1 -23279.133,E2 -23279.133} C_VEL
LIN {X 0,Y 164.408,Z 324.006,A -85,B 0,C 180,E1 -23284.693,E2 -23284.693} C_VEL
LIN {X 0,Y 164.477,Z 323.993,A -85,B 0,C 180,E1 -23290.048,E2 -23290.048} C_VEL
LIN {X 0,Y 164.518,Z 323.989,A -85,B 0,C 180,E1 -23295.149,E2 -23295.149} C_VEL
LIN {X 0,Y 164.755,Z 323.962,A -85,B 0,C 180,E1 -23300.176,E2 -23300.176} C_VEL
LIN {X 0,Y 164.811,Z 323.954,A -85,B 0,C 180,E1 -23302.65,E2 -23302.65} C_VEL
LIN {X 0,Y 165.263,Z 323.901,A -85,B 0,C 180,E1 -23310,E2 -23310} C_VEL
LIN {X 0,Y 164.811,Z 323.954,A -85,B 0,C 180,E1 -23317.35,E2 -23317.35} C_VEL
LIN {X 0,Y 164.692,Z 323.968,A -85,B 0,C 180,E1 -23321.06,E2 -23321.06} C_VEL
LIN {X 0,Y 164.494,Z 323.996,A -85,B 0,C 180,E1 -23327.402,E2 -23327.402} C_VEL
LIN {X 0,Y 164.511,Z 323.989,A -85,B 0,C 180,E1 -23329.984,E2 -23329.984} C_VEL
LIN {X 0,Y 164.385,Z 324.007,A -85,B 0,C 180,E1 -23336.136,E2 -23336.136} C_VEL
LIN {X 0,Y 164.367,Z 324.007,A -85,B 0,C 180,E1 -23341.23,E2 -23341.23} C_VEL
LIN {X 0,Y 164.286,Z 324.02,A -85,B 0,C 180,E1 -23346.792,E2 -23346.792} C_VEL
LIN {X 0,Y 164.283,Z 324.018,A -85,B 0,C 180,E1 -23349.919,E2 -23349.919} C_VEL
LIN {X 0,Y 164.272,Z 324.022,A -85,B 0,C 180,E1 -23353.344,E2 -23353.344} C_VEL
LIN {X 0,Y 164.255,Z 324.02,A -85,B 0,C 180,E1 -23356.801,E2 -23356.801} C_VEL
LIN {X 0,Y 164.294,Z 324.019,A -85,B 0,C 180,E1 -23360.353,E2 -23360.353} C_VEL
LIN {X 0,Y 164.582,Z 323.978,A -85,B 0,C 180,E1 -23366.285,E2 -23366.285} C_VEL
LIN {X 0,Y 164.772,Z 323.959,A -85,B 0,C 180,E1 -23368.546,E2 -23368.546} C_VEL
LIN {X 0,Y 164.563,Z 324.256,A -85,B 0,C 180,E1 -23369.53,E2 -23369.53} C_VEL
LIN {X 0,Y 163.807,Z 329.129,A -85,B 0,C 180,E1 -23374.597,E2 -23374.597} C_VEL
LIN {X 0,Y 163.158,Z 334.253,A -85,B 0,C 180,E1 -23379.846,E2 -23379.846} C_VEL
LIN {X 0,Y 162.661,Z 340.575,A -85,B 0,C 180,E1 -23386.256,E2 -23386.256} C_VEL
LIN {X 0,Y 163.129,Z 343.783,A -85,B 0,C 180,E1 -23389.453,E2 -23389.453} C_VEL
LIN {X 0,Y 164.512,Z 357.423,A -85,B 0,C 180,E1 -23391.404,E2 -23391.404} C_VEL
LIN {X 0,Y 164.145,Z 368.354,A -85,B 0,C 180,E1 -23393.55,E2 -23393.55} C_VEL
LIN {X 0,Y 163.805,Z 379.539,A -85,B 0,C 180,E1 -23396.313,E2 -23396.313} C_VEL
LIN {X 0,Y 163.345,Z 389.429,A -85,B 0,C 180,E1 -23399.387,E2 -23399.387} C_VEL
LIN {X 0,Y 163.364,Z 397.536,A -85,B 0,C 180,E1 -23402.469,E2 -23402.469} C_VEL
LIN {X 0,Y 164.061,Z 405.453,A -85,B 0,C 180,E1 -23406.151,E2 -23406.151} C_VEL
LIN {X 0,Y 165.546,Z 411.903,A -85,B 0,C 180,E1 -23409.78,E2 -23409.78} C_VEL
LIN {X 0,Y 167.965,Z 416.935,A -85,B 0,C 180,E1 -23413.308,E2 -23413.308} C_VEL
LIN {X 0,Y 171.232,Z 420.85,A -85,B 0,C 180,E1 -23416.7,E2 -23416.7} C_VEL
LIN {X 0,Y 173.821,Z 422.797,A -85,B 0,C 180,E1 -23418.875,E2 -23418.875} C_VEL
LIN {X 0,Y 176.758,Z 424.296,A -85,B 0,C 180,E1 -23420.971,E2 -23420.971} C_VEL
LIN {X 0,Y 180.004,Z 425.314,A -85,B 0,C 180,E1 -23422.984,E2 -23422.984} C_VEL
LIN {X 0,Y 183.542,Z 425.876,A -85,B 0,C 180,E1 -23424.913,E2 -23424.913} C_VEL
LIN {X 0,Y 187.3,Z 425.98,A -85,B 0,C 180,E1 -23426.764,E2 -23426.764} C_VEL
LIN {X 0,Y 193.745,Z 425.249,A -85,B 0,C 180,E1 -23429.472,E2 -23429.472} C_VEL
LIN {X 0,Y 199.529,Z 423.846,A -85,B 0,C 180,E1 -23431.896,E2 -23431.896} C_VEL
LIN {X 0,Y 201.948,Z 423.094,A -85,B 0,C 180,E1 -23433.839,E2 -23433.839} C_VEL
LIN {X 0,Y 204.043,Z 422.476,A -85,B 0,C 180,E1 -23435.844,E2 -23435.844} C_VEL
LIN {X 0,Y 205.668,Z 422.136,A -85,B 0,C 180,E1 -23438.192,E2 -23438.192} C_VEL
LIN {X 0,Y 206.446,Z 422.307,A -85,B 0,C 180,E1 -23440.305,E2 -23440.305} C_VEL
LIN {X 0,Y 207.016,Z 422.988,A -85,B 0,C 180,E1 -23442.767,E2 -23442.767} C_VEL
LIN {X 0,Y 207.319,Z 424.208,A -85,B 0,C 180,E1 -23445.392,E2 -23445.392} C_VEL
LIN {X 0,Y 206.87,Z 425.568,A -85,B 0,C 180,E1 -23447.198,E2 -23447.198} C_VEL
LIN {X 0,Y 203.077,Z 428.382,A -85,B 0,C 180,E1 -23448.887,E2 -23448.887} C_VEL
LIN {X 0,Y 196.278,Z 432.397,A -85,B 0,C 180,E1 -23451.199,E2 -23451.199} C_VEL
LIN {X 0,Y 189.659,Z 435.678,A -85,B 0,C 180,E1 -23453.637,E2 -23453.637} C_VEL
LIN {X 0,Y 181.911,Z 438.893,A -85,B 0,C 180,E1 -23457.256,E2 -23457.256} C_VEL
LIN {X 0,Y 175.414,Z 440.874,A -85,B 0,C 180,E1 -23461.263,E2 -23461.263} C_VEL
LIN {X 0,Y 170.276,Z 441.654,A -85,B 0,C 180,E1 -23465.623,E2 -23465.623} C_VEL
LIN {X 0,Y 166.651,Z 441.31,A -85,B 0,C 180,E1 -23470.283,E2 -23470.283} C_VEL
LIN {X 0,Y 164.654,Z 439.825,A -85,B 0,C 180,E1 -23475.161,E2 -23475.161} C_VEL
LIN {X 0,Y 164.247,Z 437.099,A -85,B 0,C 180,E1 -23480.145,E2 -23480.145} C_VEL
LIN {X 0,Y 165.257,Z 433.015,A -85,B 0,C 180,E1 -23485.121,E2 -23485.121} C_VEL
LIN {X 0,Y 166.156,Z 430.311,A -85,B 0,C 180,E1 -23487.576,E2 -23487.576} C_VEL
LIN {X 0,Y 167.298,Z 425.03,A -85,B 0,C 180,E1 -23491.204,E2 -23491.204} C_VEL
LIN {X 0,Y 168.293,Z 422.483,A -85,B 0,C 180,E1 -23492.843,E2 -23492.843} C_VEL
LIN {X 0,Y 166.474,Z 428.153,A -85,B 0,C 180,E1 -23496.058,E2 -23496.058} C_VEL
LIN {X 0,Y 165.306,Z 432.908,A -85,B 0,C 180,E1 -23499.791,E2 -23499.791} C_VEL
LIN {X 0,Y 165.047,Z 435.378,A -85,B 0,C 180,E1 -23502.293,E2 -23502.293} C_VEL
LIN {X 0,Y 165.357,Z 437.336,A -85,B 0,C 180,E1 -23504.774,E2 -23504.774} C_VEL
LIN {X 0,Y 166.137,Z 438.836,A -85,B 0,C 180,E1 -23507.225,E2 -23507.225} C_VEL
LIN {X 0,Y 167.402,Z 439.903,A -85,B 0,C 180,E1 -23509.625,E2 -23509.625} C_VEL
LIN {X 0,Y 169.205,Z 440.541,A -85,B 0,C 180,E1 -23511.951,E2 -23511.951} C_VEL
LIN {X 0,Y 171.445,Z 440.735,A -85,B 0,C 180,E1 -23514.2,E2 -23514.2} C_VEL
LIN {X 0,Y 174.083,Z 440.457,A -85,B 0,C 180,E1 -23516.365,E2 -23516.365} C_VEL
LIN {X 0,Y 177.168,Z 439.727,A -85,B 0,C 180,E1 -23518.426,E2 -23518.426} C_VEL
LIN {X 0,Y 180.662,Z 438.531,A -85,B 0,C 180,E1 -23520.379,E2 -23520.379} C_VEL
LIN {X 0,Y 186.53,Z 435.887,A -85,B 0,C 180,E1 -23523.115,E2 -23523.115} C_VEL
LIN {X 0,Y 193.115,Z 431.932,A -85,B 0,C 180,E1 -23525.612,E2 -23525.612} C_VEL
LIN {X 0,Y 197.662,Z 428.775,A -85,B 0,C 180,E1 -23527.041,E2 -23527.041} C_VEL
LIN {X 0,Y 199.733,Z 427.058,A -85,B 0,C 180,E1 -23527.858,E2 -23527.858} C_VEL
LIN {X 0,Y 201.709,Z 424.793,A -85,B 0,C 180,E1 -23529.307,E2 -23529.307} C_VEL
LIN {X 0,Y 202.653,Z 422.96,A -85,B 0,C 180,E1 -23530.891,E2 -23530.891} C_VEL
LIN {X 0,Y 202.876,Z 421.103,A -85,B 0,C 180,E1 -23533.178,E2 -23533.178} C_VEL
LIN {X 0,Y 202.485,Z 419.972,A -85,B 0,C 180,E1 -23535.508,E2 -23535.508} C_VEL
LIN {X 0,Y 202.085,Z 419.627,A -85,B 0,C 180,E1 -23536.914,E2 -23536.914} C_VEL
LIN {X 0,Y 201.443,Z 419.579,A -85,B 0,C 180,E1 -23538.477,E2 -23538.477} C_VEL
LIN {X 0,Y 200.031,Z 420.082,A -85,B 0,C 180,E1 -23540.768,E2 -23540.768} C_VEL
LIN {X 0,Y 198.071,Z 420.985,A -85,B 0,C 180,E1 -23542.898,E2 -23542.898} C_VEL
LIN {X 0,Y 195.678,Z 422.165,A -85,B 0,C 180,E1 -23544.921,E2 -23544.921} C_VEL
LIN {X 0,Y 193.113,Z 423.273,A -85,B 0,C 180,E1 -23546.911,E2 -23546.911} C_VEL
LIN {X 0,Y 189.836,Z 424.391,A -85,B 0,C 180,E1 -23548.779,E2 -23548.779} C_VEL
LIN {X 0,Y 185.461,Z 425.406,A -85,B 0,C 180,E1 -23550.483,E2 -23550.483} C_VEL
LIN {X 0,Y 181.298,Z 425.846,A -85,B 0,C 180,E1 -23552.275,E2 -23552.275} C_VEL
LIN {X 0,Y 177.342,Z 425.72,A -85,B 0,C 180,E1 -23554.153,E2 -23554.153} C_VEL
LIN {X 0,Y 173.681,Z 425.009,A -85,B 0,C 180,E1 -23556.128,E2 -23556.128} C_VEL
LIN {X 0,Y 170.331,Z 423.729,A -85,B 0,C 180,E1 -23558.198,E2 -23558.198} C_VEL
LIN {X 0,Y 165.911,Z 420.696,A -85,B 0,C 180,E1 -23561.473,E2 -23561.473} C_VEL
LIN {X 0,Y 162.258,Z 416.372,A -85,B 0,C 180,E1 -23564.934,E2 -23564.934} C_VEL
LIN {X 0,Y 159.54,Z 410.432,A -85,B 0,C 180,E1 -23568.563,E2 -23568.563} C_VEL
LIN {X 0,Y 158.061,Z 404.295,A -85,B 0,C 180,E1 -23571.688,E2 -23571.688} C_VEL
LIN {X 0,Y 157.404,Z 396.549,A -85,B 0,C 180,E1 -23574.873,E2 -23574.873} C_VEL
LIN {X 0,Y 157.372,Z 386.872,A -85,B 0,C 180,E1 -23578.077,E2 -23578.077} C_VEL
LIN {X 0,Y 157.769,Z 378.395,A -85,B 0,C 180,E1 -23580.316,E2 -23580.316} C_VEL
LIN {X 0,Y 158.181,Z 370.644,A -85,B 0,C 180,E1 -23581.906,E2 -23581.906} C_VEL
LIN {X 0,Y 158.337,Z 361.414,A -85,B 0,C 180,E1 -23583.416,E2 -23583.416} C_VEL
LIN {X 0,Y 156.267,Z 341.109,A -85,B 0,C 180,E1 -23596.994,E2 -23596.994} C_VEL
LIN {X 0,Y 156.552,Z 333.164,A -85,B 0,C 180,E1 -23602.428,E2 -23602.428} C_VEL
LIN {X 0,Y 157.091,Z 324.922,A -85,B 0,C 180,E1 -23608.105,E2 -23608.105} C_VEL
LIN {X 0,Y 157.349,Z 324.886,A -85,B 0,C 180,E1 -23609.423,E2 -23609.423} C_VEL
LIN {X 0,Y 157.334,Z 324.884,A -85,B 0,C 180,E1 -23612.41,E2 -23612.41} C_VEL
LIN {X 0,Y 157.262,Z 324.893,A -85,B 0,C 180,E1 -23616.446,E2 -23616.446} C_VEL
LIN {X 0,Y 157.184,Z 324.9,A -85,B 0,C 180,E1 -23622.114,E2 -23622.114} C_VEL
LIN {X 0,Y 157.185,Z 324.904,A -85,B 0,C 180,E1 -23627.881,E2 -23627.881} C_VEL
LIN {X 0,Y 157.26,Z 324.894,A -85,B 0,C 180,E1 -23633.548,E2 -23633.548} C_VEL
LIN {X 0,Y 157.285,Z 324.891,A -85,B 0,C 180,E1 -23638.094,E2 -23638.094} C_VEL
LIN {X 0,Y 157.314,Z 324.888,A -85,B 0,C 180,E1 -23643.464,E2 -23643.464} C_VEL
LIN {X 0,Y 157.387,Z 324.875,A -85,B 0,C 180,E1 -23649.665,E2 -23649.665} C_VEL
LIN {X 0,Y 157.45,Z 324.871,A -85,B 0,C 180,E1 -23654.465,E2 -23654.465} C_VEL
LIN {X 0,Y 157.677,Z 324.842,A -85,B 0,C 180,E1 -23659.73,E2 -23659.73} C_VEL
LIN {X 0,Y 157.749,Z 324.835,A -85,B 0,C 180,E1 -23662.319,E2 -23662.319} C_VEL
LIN {X 0,Y 158.226,Z 324.777,A -85,B 0,C 180,E1 -23670,E2 -23670} C_VEL
LIN {X 0,Y 157.749,Z 324.835,A -85,B 0,C 180,E1 -23677.681,E2 -23677.681} C_VEL
LIN {X 0,Y 157.626,Z 324.848,A -85,B 0,C 180,E1 -23681.236,E2 -23681.236} C_VEL
LIN {X 0,Y 157.452,Z 324.871,A -85,B 0,C 180,E1 -23685.534,E2 -23685.534} C_VEL
LIN {X 0,Y 157.407,Z 324.873,A -85,B 0,C 180,E1 -23690.928,E2 -23690.928} C_VEL
LIN {X 0,Y 157.307,Z 324.889,A -85,B 0,C 180,E1 -23696.687,E2 -23696.687} C_VEL
LIN {X 0,Y 157.267,Z 324.893,A -85,B 0,C 180,E1 -23702.429,E2 -23702.429} C_VEL
LIN {X 0,Y 157.26,Z 324.894,A -85,B 0,C 180,E1 -23706.452,E2 -23706.452} C_VEL
LIN {X 0,Y 157.185,Z 324.904,A -85,B 0,C 180,E1 -23712.119,E2 -23712.119} C_VEL
LIN {X 0,Y 157.186,Z 324.9,A -85,B 0,C 180,E1 -23717.886,E2 -23717.886} C_VEL
LIN {X 0,Y 157.341,Z 324.883,A -85,B 0,C 180,E1 -23723.515,E2 -23723.515} C_VEL
LIN {X 0,Y 157.653,Z 324.844,A -85,B 0,C 180,E1 -23727.887,E2 -23727.887} C_VEL
LIN {X 0,Y 157.42,Z 325.006,A -85,B 0,C 180,E1 -23729.67,E2 -23729.67} C_VEL
LIN {X 0,Y 156.647,Z 329.869,A -85,B 0,C 180,E1 -23734.929,E2 -23734.929} C_VEL
LIN {X 0,Y 156.018,Z 334.821,A -85,B 0,C 180,E1 -23740.215,E2 -23740.215} C_VEL
LIN {X 0,Y 156.202,Z 344.132,A -85,B 0,C 180,E1 -23749.977,E2 -23749.977} C_VEL
LIN {X 0,Y 157.519,Z 356.516,A -85,B 0,C 180,E1 -23751.816,E2 -23751.816} C_VEL
LIN {X 0,Y 157.233,Z 367.071,A -85,B 0,C 180,E1 -23753.91,E2 -23753.91} C_VEL
LIN {X 0,Y 156.883,Z 378.587,A -85,B 0,C 180,E1 -23756.793,E2 -23756.793} C_VEL
LIN {X 0,Y 156.511,Z 386.834,A -85,B 0,C 180,E1 -23759.36,E2 -23759.36} C_VEL
LIN {X 0,Y 156.548,Z 396.928,A -85,B 0,C 180,E1 -23763.22,E2 -23763.22} C_VEL
LIN {X 0,Y 157.348,Z 405.13,A -85,B 0,C 180,E1 -23767.059,E2 -23767.059} C_VEL
LIN {X 0,Y 159.352,Z 412.642,A -85,B 0,C 180,E1 -23771.45,E2 -23771.45} C_VEL
LIN {X 0,Y 162.114,Z 417.733,A -85,B 0,C 180,E1 -23775.08,E2 -23775.08} C_VEL
LIN {X 0,Y 165.737,Z 421.643,A -85,B 0,C 180,E1 -23778.547,E2 -23778.547} C_VEL
LIN {X 0,Y 170.131,Z 424.464,A -85,B 0,C 180,E1 -23781.829,E2 -23781.829} C_VEL
LIN {X 0,Y 173.498,Z 425.768,A -85,B 0,C 180,E1 -23783.899,E2 -23783.899} C_VEL
LIN {X 0,Y 177.138,Z 426.614,A -85,B 0,C 180,E1 -23785.879,E2 -23785.879} C_VEL
LIN {X 0,Y 181.035,Z 427.012,A -85,B 0,C 180,E1 -23787.768,E2 -23787.768} C_VEL
LIN {X 0,Y 187.533,Z 426.779,A -85,B 0,C 180,E1 -23790.464,E2 -23790.464} C_VEL
LIN {X 0,Y 193.665,Z 425.771,A -85,B 0,C 180,E1 -23792.983,E2 -23792.983} C_VEL
LIN {X 0,Y 196.156,Z 425.341,A -85,B 0,C 180,E1 -23794.981,E2 -23794.981} C_VEL
LIN {X 0,Y 198.185,Z 425.025,A -85,B 0,C 180,E1 -23797.077,E2 -23797.077} C_VEL
LIN {X 0,Y 199.55,Z 425.076,A -85,B 0,C 180,E1 -23799.345,E2 -23799.345} C_VEL
LIN {X 0,Y 200.534,Z 425.866,A -85,B 0,C 180,E1 -23802.61,E2 -23802.61} C_VEL
LIN {X 0,Y 200.757,Z 426.609,A -85,B 0,C 180,E1 -23804.442,E2 -23804.442} C_VEL
LIN {X 0,Y 200.704,Z 427.24,A -85,B 0,C 180,E1 -23805.546,E2 -23805.546} C_VEL
LIN {X 0,Y 199.851,Z 428.259,A -85,B 0,C 180,E1 -23806.706,E2 -23806.706} C_VEL
LIN {X 0,Y 195.562,Z 430.736,A -85,B 0,C 180,E1 -23808.329,E2 -23808.329} C_VEL
LIN {X 0,Y 188.478,Z 434.087,A -85,B 0,C 180,E1 -23810.661,E2 -23810.661} C_VEL
LIN {X 0,Y 179.896,Z 437.389,A -85,B 0,C 180,E1 -23814.126,E2 -23814.126} C_VEL
LIN {X 0,Y 172.412,Z 439.5,A -85,B 0,C 180,E1 -23818,E2 -23818} C_VEL
LIN {X 0,Y 166.398,Z 440.434,A -85,B 0,C 180,E1 -23822.316,E2 -23822.316} C_VEL
LIN {X 0,Y 161.808,Z 440.238,A -85,B 0,C 180,E1 -23826.989,E2 -23826.989} C_VEL
LIN {X 0,Y 158.862,Z 438.965,A -85,B 0,C 180,E1 -23831.96,E2 -23831.96} C_VEL
LIN {X 0,Y 157.582,Z 436.538,A -85,B 0,C 180,E1 -23837.115,E2 -23837.115} C_VEL
LIN {X 0,Y 157.953,Z 432.833,A -85,B 0,C 180,E1 -23842.329,E2 -23842.329} C_VEL
LIN {X 0,Y 159.123,Z 429.055,A -85,B 0,C 180,E1 -23846.201,E2 -23846.201} C_VEL
LIN {X 0,Y 159.993,Z 425.857,A -85,B 0,C 180,E1 -23848.741,E2 -23848.741} C_VEL
LIN {X 0,Y 161.841,Z 419.448,A -85,B 0,C 180,E1 -23852.776,E2 -23852.776} C_VEL
LIN {X 0,Y 162.088,Z 419.066,A -85,B 0,C 180,E1 -23853.037,E2 -23853.037} C_VEL
LIN {X 0,Y 160.511,Z 423.869,A -85,B 0,C 180,E1 -23855.654,E2 -23855.654} C_VEL
LIN {X 0,Y 159.218,Z 428.534,A -85,B 0,C 180,E1 -23858.887,E2 -23858.887} C_VEL
LIN {X 0,Y 158.566,Z 432.856,A -85,B 0,C 180,E1 -23862.804,E2 -23862.804} C_VEL
LIN {X 0,Y 158.83,Z 435.073,A -85,B 0,C 180,E1 -23865.396,E2 -23865.396} C_VEL
LIN {X 0,Y 159.638,Z 436.819,A -85,B 0,C 180,E1 -23867.949,E2 -23867.949} C_VEL
LIN {X 0,Y 160.928,Z 438.107,A -85,B 0,C 180,E1 -23870.449,E2 -23870.449} C_VEL
LIN {X 0,Y 162.789,Z 439.02,A -85,B 0,C 180,E1 -23872.865,E2 -23872.865} C_VEL
LIN {X 0,Y 165.081,Z 439.492,A -85,B 0,C 180,E1 -23875.197,E2 -23875.197} C_VEL
LIN {X 0,Y 167.813,Z 439.563,A -85,B 0,C 180,E1 -23877.431,E2 -23877.431} C_VEL
LIN {X 0,Y 170.979,Z 439.2,A -85,B 0,C 180,E1 -23879.555,E2 -23879.555} C_VEL
LIN {X 0,Y 174.593,Z 438.369,A -85,B 0,C 180,E1 -23881.554,E2 -23881.554} C_VEL
LIN {X 0,Y 178.534,Z 437.048,A -85,B 0,C 180,E1 -23883.444,E2 -23883.444} C_VEL
LIN {X 0,Y 185.066,Z 434.181,A -85,B 0,C 180,E1 -23886.06,E2 -23886.06} C_VEL
LIN {X 0,Y 192.831,Z 429.722,A -85,B 0,C 180,E1 -23888.543,E2 -23888.543} C_VEL
LIN {X 0,Y 199.452,Z 424.859,A -85,B 0,C 180,E1 -23890.684,E2 -23890.684} C_VEL
LIN {X 0,Y 201.371,Z 423.004,A -85,B 0,C 180,E1 -23891.538,E2 -23891.538} C_VEL
LIN {X 0,Y 203.069,Z 421.289,A -85,B 0,C 180,E1 -23892.493,E2 -23892.493} C_VEL
LIN {X 0,Y 202.944,Z 420.524,A -85,B 0,C 180,E1 -23893.837,E2 -23893.837} C_VEL
LIN {X 0,Y 202.485,Z 419.972,A -85,B 0,C 180,E1 -23895.508,E2 -23895.508} C_VEL
LIN {X 0,Y 201.897,Z 419.885,A -85,B 0,C 180,E1 -23896.607,E2 -23896.607} C_VEL
LIN {X 0,Y 200.045,Z 420.566,A -85,B 0,C 180,E1 -23898.2,E2 -23898.2} C_VEL
LIN {X 0,Y 197.476,Z 421.712,A -85,B 0,C 180,E1 -23899.722,E2 -23899.722} C_VEL
LIN {X 0,Y 191.562,Z 424.197,A -85,B 0,C 180,E1 -23902.841,E2 -23902.841} C_VEL
LIN {X 0,Y 189.825,Z 424.738,A -85,B 0,C 180,E1 -23903.952,E2 -23903.952} C_VEL
LIN {X 0,Y 187.392,Z 425.391,A -85,B 0,C 180,E1 -23905.764,E2 -23905.764} C_VEL
LIN {X 0,Y 183.895,Z 426.127,A -85,B 0,C 180,E1 -23907.65,E2 -23907.65} C_VEL
LIN {X 0,Y 179.37,Z 426.756,A -85,B 0,C 180,E1 -23909.376,E2 -23909.376} C_VEL
LIN {X 0,Y 175.071,Z 426.814,A -85,B 0,C 180,E1 -23911.199,E2 -23911.199} C_VEL
LIN {X 0,Y 170.972,Z 426.306,A -85,B 0,C 180,E1 -23913.114,E2 -23913.114} C_VEL
LIN {X 0,Y 167.211,Z 425.23,A -85,B 0,C 180,E1 -23915.143,E2 -23915.143} C_VEL
LIN {X 0,Y 162.137,Z 422.602,A -85,B 0,C 180,E1 -23918.377,E2 -23918.377} C_VEL
LIN {X 0,Y 157.852,Z 418.559,A -85,B 0,C 180,E1 -23921.838,E2 -23921.838} C_VEL
LIN {X 0,Y 154.441,Z 413.171,A -85,B 0,C 180,E1 -23925.502,E2 -23925.502} C_VEL
LIN {X 0,Y 152.388,Z 407.378,A -85,B 0,C 180,E1 -23928.693,E2 -23928.693} C_VEL
LIN {X 0,Y 151.14,Z 400.348,A -85,B 0,C 180,E1 -23931.978,E2 -23931.978} C_VEL
LIN {X 0,Y 150.664,Z 391.606,A -85,B 0,C 180,E1 -23935.314,E2 -23935.314} C_VEL
LIN {X 0,Y 150.875,Z 382.813,A -85,B 0,C 180,E1 -23937.994,E2 -23937.994} C_VEL
LIN {X 0,Y 151.388,Z 373.237,A -85,B 0,C 180,E1 -23940.329,E2 -23940.329} C_VEL
LIN {X 0,Y 151.715,Z 362.883,A -85,B 0,C 180,E1 -23942.154,E2 -23942.154} C_VEL
LIN {X 0,Y 151.671,Z 362.107,A -85,B 0,C 180,E1 -23942.32,E2 -23942.32} C_VEL
LIN {X 0,Y 149.149,Z 341.673,A -85,B 0,C 180,E1 -23956.419,E2 -23956.419} C_VEL
LIN {X 0,Y 149.435,Z 333.643,A -85,B 0,C 180,E1 -23962.097,E2 -23962.097} C_VEL
LIN {X 0,Y 149.949,Z 325.812,A -85,B 0,C 180,E1 -23967.649,E2 -23967.649} C_VEL
LIN {X 0,Y 150.274,Z 325.766,A -85,B 0,C 180,E1 -23970.956,E2 -23970.956} C_VEL
LIN {X 0,Y 150.214,Z 325.766,A -85,B 0,C 180,E1 -23974.151,E2 -23974.151} C_VEL
LIN {X 0,Y 150.166,Z 325.78,A -85,B 0,C 180,E1 -23977.471,E2 -23977.471} C_VEL
LIN {X 0,Y 150.127,Z 325.78,A -85,B 0,C 180,E1 -23981.494,E2 -23981.494} C_VEL
LIN {X 0,Y 150.119,Z 325.785,A -85,B 0,C 180,E1 -23985.393,E2 -23985.393} C_VEL
LIN {X 0,Y 150.134,Z 325.782,A -85,B 0,C 180,E1 -23989.053,E2 -23989.053} C_VEL
LIN {X 0,Y 150.171,Z 325.775,A -85,B 0,C 180,E1 -23992.705,E2 -23992.705} C_VEL
LIN {X 0,Y 150.207,Z 325.773,A -85,B 0,C 180,E1 -23997.365,E2 -23997.365} C_VEL
LIN {X 0,Y 150.236,Z 325.771,A -85,B 0,C 180,E1 -24002.716,E2 -24002.716} C_VEL
LIN {X 0,Y 150.343,Z 325.753,A -85,B 0,C 180,E1 -24009.205,E2 -24009.205} C_VEL
LIN {X 0,Y 150.359,Z 325.755,A -85,B 0,C 180,E1 -24013.713,E2 -24013.713} C_VEL
LIN {X 0,Y 150.6,Z 325.723,A -85,B 0,C 180,E1 -24019.242,E2 -24019.242} C_VEL
LIN {X 0,Y 150.688,Z 325.715,A -85,B 0,C 180,E1 -24021.957,E2 -24021.957} C_VEL
LIN {X 0,Y 151.186,Z 325.654,A -85,B 0,C 180,E1 -24030,E2 -24030} C_VEL
LIN {X 0,Y 150.688,Z 325.715,A -85,B 0,C 180,E1 -24038.043,E2 -24038.043} C_VEL
LIN {X 0,Y 150.567,Z 325.727,A -85,B 0,C 180,E1 -24041.436,E2 -24041.436} C_VEL
LIN {X 0,Y 150.365,Z 325.754,A -85,B 0,C 180,E1 -24046.286,E2 -24046.286} C_VEL
LIN {X 0,Y 150.381,Z 325.748,A -85,B 0,C 180,E1 -24050.833,E2 -24050.833} C_VEL
LIN {X 0,Y 150.236,Z 325.771,A -85,B 0,C 180,E1 -24057.284,E2 -24057.284} C_VEL
LIN {X 0,Y 150.207,Z 325.773,A -85,B 0,C 180,E1 -24062.635,E2 -24062.635} C_VEL
LIN {X 0,Y 150.165,Z 325.775,A -85,B 0,C 180,E1 -24067.476,E2 -24067.476} C_VEL
LIN {X 0,Y 150.129,Z 325.784,A -85,B 0,C 180,E1 -24071.501,E2 -24071.501} C_VEL
LIN {X 0,Y 150.119,Z 325.782,A -85,B 0,C 180,E1 -24075.398,E2 -24075.398} C_VEL
LIN {X 0,Y 150.137,Z 325.782,A -85,B 0,C 180,E1 -24079.059,E2 -24079.059} C_VEL
LIN {X 0,Y 150.232,Z 325.772,A -85,B 0,C 180,E1 -24082.682,E2 -24082.682} C_VEL
LIN {X 0,Y 150.536,Z 325.732,A -85,B 0,C 180,E1 -24087.178,E2 -24087.178} C_VEL
LIN {X 0,Y 150.307,Z 325.793,A -85,B 0,C 180,E1 -24089.926,E2 -24089.926} C_VEL
LIN {X 0,Y 149.345,Z 331.596,A -85,B 0,C 180,E1 -24096.426,E2 -24096.426} C_VEL
LIN {X 0,Y 148.711,Z 336.748,A -85,B 0,C 180,E1 -24102.159,E2 -24102.159} C_VEL
LIN {X 0,Y 149.328,Z 344.576,A -85,B 0,C 180,E1 -24110.649,E2 -24110.649} C_VEL
LIN {X 0,Y 150.563,Z 355.669,A -85,B 0,C 180,E1 -24112.291,E2 -24112.291} C_VEL
LIN {X 0,Y 150.34,Z 365.673,A -85,B 0,C 180,E1 -24114.302,E2 -24114.302} C_VEL
LIN {X 0,Y 150.091,Z 376.28,A -85,B 0,C 180,E1 -24116.984,E2 -24116.984} C_VEL
LIN {X 0,Y 149.694,Z 385.814,A -85,B 0,C 180,E1 -24120.003,E2 -24120.003} C_VEL
LIN {X 0,Y 149.7,Z 394.659,A -85,B 0,C 180,E1 -24123.368,E2 -24123.368} C_VEL
LIN {X 0,Y 150.473,Z 403.298,A -85,B 0,C 180,E1 -24127.383,E2 -24127.383} C_VEL
LIN {X 0,Y 152.487,Z 411.379,A -85,B 0,C 180,E1 -24131.973,E2 -24131.973} C_VEL
LIN {X 0,Y 155.306,Z 416.858,A -85,B 0,C 180,E1 -24135.758,E2 -24135.758} C_VEL
LIN {X 0,Y 159.017,Z 421.206,A -85,B 0,C 180,E1 -24139.361,E2 -24139.361} C_VEL
LIN {X 0,Y 163.543,Z 424.432,A -85,B 0,C 180,E1 -24142.756,E2 -24142.756} C_VEL
LIN {X 0,Y 167.023,Z 426.023,A -85,B 0,C 180,E1 -24144.887,E2 -24144.887} C_VEL
LIN {X 0,Y 170.78,Z 427.157,A -85,B 0,C 180,E1 -24146.919,E2 -24146.919} C_VEL
LIN {X 0,Y 174.806,Z 427.855,A -85,B 0,C 180,E1 -24148.849,E2 -24148.849} C_VEL
LIN {X 0,Y 181.605,Z 428.078,A -85,B 0,C 180,E1 -24151.637,E2 -24151.637} C_VEL
LIN {X 0,Y 187.837,Z 427.518,A -85,B 0,C 180,E1 -24154.144,E2 -24154.144} C_VEL
LIN {X 0,Y 190.303,Z 427.388,A -85,B 0,C 180,E1 -24156.223,E2 -24156.223} C_VEL
LIN {X 0,Y 192.205,Z 427.416,A -85,B 0,C 180,E1 -24158.437,E2 -24158.437} C_VEL
LIN {X 0,Y 193.336,Z 427.828,A -85,B 0,C 180,E1 -24160.871,E2 -24160.871} C_VEL
LIN {X 0,Y 193.97,Z 428.723,A -85,B 0,C 180,E1 -24163.56,E2 -24163.56} C_VEL
LIN {X 0,Y 192.675,Z 430.403,A -85,B 0,C 180,E1 -24166.128,E2 -24166.128} C_VEL
LIN {X 0,Y 187.921,Z 432.555,A -85,B 0,C 180,E1 -24167.687,E2 -24167.687} C_VEL
LIN {X 0,Y 178.45,Z 435.925,A -85,B 0,C 180,E1 -24170.939,E2 -24170.939} C_VEL
LIN {X 0,Y 170.167,Z 438.115,A -85,B 0,C 180,E1 -24174.675,E2 -24174.675} C_VEL
LIN {X 0,Y 163.176,Z 439.18,A -85,B 0,C 180,E1 -24178.879,E2 -24178.879} C_VEL
LIN {X 0,Y 157.615,Z 439.12,A -85,B 0,C 180,E1 -24183.519,E2 -24183.519} C_VEL
LIN {X 0,Y 153.659,Z 437.997,A -85,B 0,C 180,E1 -24188.537,E2 -24188.537} C_VEL
LIN {X 0,Y 151.437,Z 435.807,A -85,B 0,C 180,E1 -24193.832,E2 -24193.832} C_VEL
LIN {X 0,Y 150.98,Z 432.429,A -85,B 0,C 180,E1 -24199.269,E2 -24199.269} C_VEL
LIN {X 0,Y 152.151,Z 427.675,A -85,B 0,C 180,E1 -24204.699,E2 -24204.699} C_VEL
LIN {X 0,Y 153.14,Z 424.635,A -85,B 0,C 180,E1 -24207.37,E2 -24207.37} C_VEL
LIN {X 0,Y 154.681,Z 418.288,A -85,B 0,C 180,E1 -24211.566,E2 -24211.566} C_VEL
LIN {X 0,Y 156.023,Z 415.484,A -85,B 0,C 180,E1 -24213.334,E2 -24213.334} C_VEL
LIN {X 0,Y 154.416,Z 420.28,A -85,B 0,C 180,E1 -24215.878,E2 -24215.878} C_VEL
LIN {X 0,Y 152.932,Z 425.385,A -85,B 0,C 180,E1 -24219.256,E2 -24219.256} C_VEL
LIN {X 0,Y 152.209,Z 430.048,A -85,B 0,C 180,E1 -24223.348,E2 -24223.348} C_VEL
LIN {X 0,Y 152.784,Z 433.586,A -85,B 0,C 180,E1 -24227.397,E2 -24227.397} C_VEL
LIN {X 0,Y 154.553,Z 436.17,A -85,B 0,C 180,E1 -24231.333,E2 -24231.333} C_VEL
LIN {X 0,Y 156.447,Z 437.319,A -85,B 0,C 180,E1 -24233.848,E2 -24233.848} C_VEL
LIN {X 0,Y 158.806,Z 438.063,A -85,B 0,C 180,E1 -24236.267,E2 -24236.267} C_VEL
LIN {X 0,Y 161.638,Z 438.407,A -85,B 0,C 180,E1 -24238.573,E2 -24238.573} C_VEL
LIN {X 0,Y 164.893,Z 438.349,A -85,B 0,C 180,E1 -24240.761,E2 -24240.761} C_VEL
LIN {X 0,Y 168.604,Z 437.879,A -85,B 0,C 180,E1 -24242.812,E2 -24242.812} C_VEL
LIN {X 0,Y 172.665,Z 436.968,A -85,B 0,C 180,E1 -24244.739,E2 -24244.739} C_VEL
LIN {X 0,Y 177.039,Z 435.574,A -85,B 0,C 180,E1 -24246.546,E2 -24246.546} C_VEL
LIN {X 0,Y 184.261,Z 432.504,A -85,B 0,C 180,E1 -24249.001,E2 -24249.001} C_VEL
LIN {X 0,Y 191.843,Z 428.315,A -85,B 0,C 180,E1 -24251.255,E2 -24251.255} C_VEL
LIN {X 0,Y 194.262,Z 426.702,A -85,B 0,C 180,E1 -24252.013,E2 -24252.013} C_VEL
LIN {X 0,Y 196.319,Z 425.122,A -85,B 0,C 180,E1 -24252.858,E2 -24252.858} C_VEL
LIN {X 0,Y 196.721,Z 424.041,A -85,B 0,C 180,E1 -24254.393,E2 -24254.393} C_VEL
LIN {X 0,Y 195.933,Z 423.321,A -85,B 0,C 180,E1 -24257.034,E2 -24257.034} C_VEL
LIN {X 0,Y 194.552,Z 423.371,A -85,B 0,C 180,E1 -24259.438,E2 -24259.438} C_VEL
LIN {X 0,Y 192.616,Z 423.856,A -85,B 0,C 180,E1 -24261.66,E2 -24261.66} C_VEL
LIN {X 0,Y 189.825,Z 424.738,A -85,B 0,C 180,E1 -24263.952,E2 -24263.952} C_VEL
LIN {X 0,Y 187.636,Z 425.41,A -85,B 0,C 180,E1 -24264.917,E2 -24264.917} C_VEL
LIN {X 0,Y 184.601,Z 426.28,A -85,B 0,C 180,E1 -24265.675,E2 -24265.675} C_VEL
LIN {X 0,Y 176.499,Z 427.76,A -85,B 0,C 180,E1 -24267.238,E2 -24267.238} C_VEL
LIN {X 0,Y 173.468,Z 427.913,A -85,B 0,C 180,E1 -24268.142,E2 -24268.142} C_VEL
LIN {X 0,Y 168.879,Z 427.59,A -85,B 0,C 180,E1 -24270.037,E2 -24270.037} C_VEL
LIN {X 0,Y 164.671,Z 426.703,A -85,B 0,C 180,E1 -24271.997,E2 -24271.997} C_VEL
LIN {X 0,Y 158.962,Z 424.299,A -85,B 0,C 180,E1 -24275.161,E2 -24275.161} C_VEL
LIN {X 0,Y 154.001,Z 420.66,A -85,B 0,C 180,E1 -24278.584,E2 -24278.584} C_VEL
LIN {X 0,Y 149.923,Z 415.621,A -85,B 0,C 180,E1 -24282.256,E2 -24282.256} C_VEL
LIN {X 0,Y 146.825,Z 409.028,A -85,B 0,C 180,E1 -24286.149,E2 -24286.149} C_VEL
LIN {X 0,Y 145.125,Z 402.268,A -85,B 0,C 180,E1 -24289.533,E2 -24289.533} C_VEL
LIN {X 0,Y 144.317,Z 393.828,A -85,B 0,C 180,E1 -24293.004,E2 -24293.004} C_VEL
LIN {X 0,Y 144.283,Z 384.49,A -85,B 0,C 180,E1 -24296.156,E2 -24296.156} C_VEL
LIN {X 0,Y 144.668,Z 375.294,A -85,B 0,C 180,E1 -24298.605,E2 -24298.605} C_VEL
LIN {X 0,Y 145.064,Z 366.714,A -85,B 0,C 180,E1 -24300.343,E2 -24300.343} C_VEL
LIN {X 0,Y 145.116,Z 362.86,A -85,B 0,C 180,E1 -24301.037,E2 -24301.037} C_VEL
LIN {X 0,Y 142.099,Z 340.173,A -85,B 0,C 180,E1 -24317.258,E2 -24317.258} C_VEL
LIN {X 0,Y 142.421,Z 332.002,A -85,B 0,C 180,E1 -24323.248,E2 -24323.248} C_VEL
LIN {X 0,Y 142.818,Z 326.699,A -85,B 0,C 180,E1 -24327.213,E2 -24327.213} C_VEL
LIN {X 0,Y 143.053,Z 326.667,A -85,B 0,C 180,E1 -24329.421,E2 -24329.421} C_VEL
LIN {X 0,Y 143.2,Z 326.642,A -85,B 0,C 180,E1 -24333.453,E2 -24333.453} C_VEL
LIN {X 0,Y 143.047,Z 326.665,A -85,B 0,C 180,E1 -24339.69,E2 -24339.69} C_VEL
LIN {X 0,Y 143.027,Z 326.664,A -85,B 0,C 180,E1 -24343.461,E2 -24343.461} C_VEL
LIN {X 0,Y 143.032,Z 326.668,A -85,B 0,C 180,E1 -24347.473,E2 -24347.473} C_VEL
LIN {X 0,Y 143.067,Z 326.658,A -85,B 0,C 180,E1 -24351.805,E2 -24351.805} C_VEL
LIN {X 0,Y 143.174,Z 326.649,A -85,B 0,C 180,E1 -24357.319,E2 -24357.319} C_VEL
LIN {X 0,Y 143.182,Z 326.647,A -85,B 0,C 180,E1 -24362.061,E2 -24362.061} C_VEL
LIN {X 0,Y 143.269,Z 326.633,A -85,B 0,C 180,E1 -24368.743,E2 -24368.743} C_VEL
LIN {X 0,Y 143.297,Z 326.635,A -85,B 0,C 180,E1 -24372.886,E2 -24372.886} C_VEL
LIN {X 0,Y 143.526,Z 326.605,A -85,B 0,C 180,E1 -24378.705,E2 -24378.705} C_VEL
LIN {X 0,Y 143.61,Z 326.596,A -85,B 0,C 180,E1 -24381.558,E2 -24381.558} C_VEL
LIN {X 0,Y 144.145,Z 326.531,A -85,B 0,C 180,E1 -24390,E2 -24390} C_VEL
LIN {X 0,Y 143.61,Z 326.596,A -85,B 0,C 180,E1 -24398.442,E2 -24398.442} C_VEL
LIN {X 0,Y 143.495,Z 326.607,A -85,B 0,C 180,E1 -24401.629,E2 -24401.629} C_VEL
LIN {X 0,Y 143.309,Z 326.633,A -85,B 0,C 180,E1 -24407.112,E2 -24407.112} C_VEL
LIN {X 0,Y 143.302,Z 326.629,A -85,B 0,C 180,E1 -24411.291,E2 -24411.291} C_VEL
LIN {X 0,Y 143.182,Z 326.647,A -85,B 0,C 180,E1 -24417.939,E2 -24417.939} C_VEL
LIN {X 0,Y 143.156,Z 326.654,A -85,B 0,C 180,E1 -24423.435,E2 -24423.435} C_VEL
LIN {X 0,Y 143.048,Z 326.663,A -85,B 0,C 180,E1 -24429.695,E2 -24429.695} C_VEL
LIN {X 0,Y 143.027,Z 326.668,A -85,B 0,C 180,E1 -24433.466,E2 -24433.466} C_VEL
LIN {X 0,Y 143.033,Z 326.663,A -85,B 0,C 180,E1 -24437.479,E2 -24437.479} C_VEL
LIN {X 0,Y 143.209,Z 326.643,A -85,B 0,C 180,E1 -24443.926,E2 -24443.926} C_VEL
LIN {X 0,Y 143.483,Z 326.609,A -85,B 0,C 180,E1 -24447.403,E2 -24447.403} C_VEL
LIN {X 0,Y 143.237,Z 326.645,A -85,B 0,C 180,E1 -24449.811,E2 -24449.811} C_VEL
LIN {X 0,Y 143.072,Z 326.885,A -85,B 0,C 180,E1 -24450.584,E2 -24450.584} C_VEL
LIN {X 0,Y 142.211,Z 332.12,A -85,B 0,C 180,E1 -24456.716,E2 -24456.716} C_VEL
LIN {X 0,Y 141.686,Z 336.246,A -85,B 0,C 180,E1 -24461.494,E2 -24461.494} C_VEL
LIN {X 0,Y 142.309,Z 344.579,A -85,B 0,C 180,E1 -24471.009,E2 -24471.009} C_VEL
LIN {X 0,Y 142.455,Z 344.862,A -85,B 0,C 180,E1 -24471.32,E2 -24471.32} C_VEL
LIN {X 0,Y 143.698,Z 355.503,A -85,B 0,C 180,E1 -24472.981,E2 -24472.981} C_VEL
LIN {X 0,Y 143.461,Z 365.398,A -85,B 0,C 180,E1 -24475.086,E2 -24475.086} C_VEL
LIN {X 0,Y 143.241,Z 376.07,A -85,B 0,C 180,E1 -24477.895,E2 -24477.895} C_VEL
LIN {X 0,Y 142.856,Z 386.686,A -85,B 0,C 180,E1 -24481.413,E2 -24481.413} C_VEL
LIN {X 0,Y 143.064,Z 395.331,A -85,B 0,C 180,E1 -24484.935,E2 -24484.935} C_VEL
LIN {X 0,Y 144.066,Z 403.917,A -85,B 0,C 180,E1 -24489.126,E2 -24489.126} C_VEL
LIN {X 0,Y 146.09,Z 410.929,A -85,B 0,C 180,E1 -24493.213,E2 -24493.213} C_VEL
LIN {X 0,Y 149.731,Z 417.497,A -85,B 0,C 180,E1 -24497.767,E2 -24497.767} C_VEL
LIN {X 0,Y 153.833,Z 421.882,A -85,B 0,C 180,E1 -24501.441,E2 -24501.441} C_VEL
LIN {X 0,Y 157.006,Z 424.187,A -85,B 0,C 180,E1 -24503.761,E2 -24503.761} C_VEL
LIN {X 0,Y 160.583,Z 426.081,A -85,B 0,C 180,E1 -24505.958,E2 -24505.958} C_VEL
LIN {X 0,Y 164.472,Z 427.493,A -85,B 0,C 180,E1 -24508.04,E2 -24508.04} C_VEL
LIN {X 0,Y 168.628,Z 428.489,A -85,B 0,C 180,E1 -24510.012,E2 -24510.012} C_VEL
LIN {X 0,Y 175.876,Z 429.186,A -85,B 0,C 180,E1 -24512.948,E2 -24512.948} C_VEL
LIN {X 0,Y 177.73,Z 429.176,A -85,B 0,C 180,E1 -24513.618,E2 -24513.618} C_VEL
LIN {X 0,Y 181.998,Z 429.075,A -85,B 0,C 180,E1 -24515.4,E2 -24515.4} C_VEL
LIN {X 0,Y 184.368,Z 429.237,A -85,B 0,C 180,E1 -24517.586,E2 -24517.586} C_VEL
LIN {X 0,Y 186.081,Z 429.6,A -85,B 0,C 180,E1 -24519.949,E2 -24519.949} C_VEL
LIN {X 0,Y 186.581,Z 429.892,A -85,B 0,C 180,E1 -24521.119,E2 -24521.119} C_VEL
LIN {X 0,Y 186.894,Z 430.417,A -85,B 0,C 180,E1 -24522.603,E2 -24522.603} C_VEL
LIN {X 0,Y 186.603,Z 431.215,A -85,B 0,C 180,E1 -24524.308,E2 -24524.308} C_VEL
LIN {X 0,Y 182.738,Z 432.949,A -85,B 0,C 180,E1 -24526.19,E2 -24526.19} C_VEL
LIN {X 0,Y 173.015,Z 435.765,A -85,B 0,C 180,E1 -24529.463,E2 -24529.463} C_VEL
LIN {X 0,Y 164.467,Z 437.448,A -85,B 0,C 180,E1 -24533.255,E2 -24533.255} C_VEL
LIN {X 0,Y 157.212,Z 438.053,A -85,B 0,C 180,E1 -24537.558,E2 -24537.558} C_VEL
LIN {X 0,Y 151.404,Z 437.572,A -85,B 0,C 180,E1 -24542.342,E2 -24542.342} C_VEL
LIN {X 0,Y 147.293,Z 436.077,A -85,B 0,C 180,E1 -24547.56,E2 -24547.56} C_VEL
LIN {X 0,Y 144.947,Z 433.526,A -85,B 0,C 180,E1 -24553.087,E2 -24553.087} C_VEL
LIN {X 0,Y 144.475,Z 429.84,A -85,B 0,C 180,E1 -24558.78,E2 -24558.78} C_VEL
LIN {X 0,Y 145.716,Z 424.735,A -85,B 0,C 180,E1 -24564.465,E2 -24564.465} C_VEL
LIN {X 0,Y 146.754,Z 421.497,A -85,B 0,C 180,E1 -24567.255,E2 -24567.255} C_VEL
LIN {X 0,Y 148.455,Z 414.804,A -85,B 0,C 180,E1 -24571.632,E2 -24571.632} C_VEL
LIN {X 0,Y 150.099,Z 411.658,A -85,B 0,C 180,E1 -24573.639,E2 -24573.639} C_VEL
LIN {X 0,Y 148.103,Z 417.471,A -85,B 0,C 180,E1 -24576.676,E2 -24576.676} C_VEL
LIN {X 0,Y 146.831,Z 421.926,A -85,B 0,C 180,E1 -24579.644,E2 -24579.644} C_VEL
LIN {X 0,Y 145.982,Z 427.016,A -85,B 0,C 180,E1 -24583.929,E2 -24583.929} C_VEL
LIN {X 0,Y 146.475,Z 430.991,A -85,B 0,C 180,E1 -24588.172,E2 -24588.172} C_VEL
LIN {X 0,Y 148.312,Z 433.875,A -85,B 0,C 180,E1 -24592.278,E2 -24592.278} C_VEL
LIN {X 0,Y 150.225,Z 435.353,A -85,B 0,C 180,E1 -24594.901,E2 -24594.901} C_VEL
LIN {X 0,Y 152.654,Z 436.414,A -85,B 0,C 180,E1 -24597.412,E2 -24597.412} C_VEL
LIN {X 0,Y 155.549,Z 437.057,A -85,B 0,C 180,E1 -24599.802,E2 -24599.802} C_VEL
LIN {X 0,Y 158.904,Z 437.293,A -85,B 0,C 180,E1 -24602.055,E2 -24602.055} C_VEL
LIN {X 0,Y 162.715,Z 437.134,A -85,B 0,C 180,E1 -24604.159,E2 -24604.159} C_VEL
LIN {X 0,Y 166.893,Z 436.56,A -85,B 0,C 180,E1 -24606.125,E2 -24606.125} C_VEL
LIN {X 0,Y 171.385,Z 435.553,A -85,B 0,C 180,E1 -24607.96,E2 -24607.96} C_VEL
LIN {X 0,Y 176.255,Z 434.09,A -85,B 0,C 180,E1 -24609.642,E2 -24609.642} C_VEL
LIN {X 0,Y 184.065,Z 430.898,A -85,B 0,C 180,E1 -24611.928,E2 -24611.928} C_VEL
LIN {X 0,Y 189.134,Z 428.238,A -85,B 0,C 180,E1 -24613.428,E2 -24613.428} C_VEL
LIN {X 0,Y 190.319,Z 427.156,A -85,B 0,C 180,E1 -24614.558,E2 -24614.558} C_VEL
LIN {X 0,Y 190.117,Z 426.884,A -85,B 0,C 180,E1 -24615.38,E2 -24615.38} C_VEL
LIN {X 0,Y 188.806,Z 426.409,A -85,B 0,C 180,E1 -24618.114,E2 -24618.114} C_VEL
LIN {X 0,Y 187.049,Z 426.514,A -85,B 0,C 180,E1 -24620.299,E2 -24620.299} C_VEL
LIN {X 0,Y 183.636,Z 427.006,A -85,B 0,C 180,E1 -24623.1,E2 -24623.1} C_VEL
LIN {X 0,Y 181.681,Z 427.253,A -85,B 0,C 180,E1 -24624.529,E2 -24624.529} C_VEL
LIN {X 0,Y 178.004,Z 427.686,A -85,B 0,C 180,E1 -24626.441,E2 -24626.441} C_VEL
LIN {X 0,Y 173.468,Z 427.913,A -85,B 0,C 180,E1 -24628.142,E2 -24628.142} C_VEL
LIN {X 0,Y 169.245,Z 427.788,A -85,B 0,C 180,E1 -24629.527,E2 -24629.527} C_VEL
LIN {X 0,Y 164.494,Z 427.287,A -85,B 0,C 180,E1 -24630.747,E2 -24630.747} C_VEL
LIN {X 0,Y 158.093,Z 425.901,A -85,B 0,C 180,E1 -24632.35,E2 -24632.35} C_VEL
LIN {X 0,Y 153.766,Z 424.327,A -85,B 0,C 180,E1 -24633.723,E2 -24633.723} C_VEL
LIN {X 0,Y 150.428,Z 422.316,A -85,B 0,C 180,E1 -24635.385,E2 -24635.385} C_VEL
LIN {X 0,Y 145.954,Z 417.865,A -85,B 0,C 180,E1 -24638.826,E2 -24638.826} C_VEL
LIN {X 0,Y 142.112,Z 411.76,A -85,B 0,C 180,E1 -24642.735,E2 -24642.735} C_VEL
LIN {X 0,Y 139.784,Z 405.35,A -85,B 0,C 180,E1 -24646.179,E2 -24646.179} C_VEL
LIN {X 0,Y 138.359,Z 397.643,A -85,B 0,C 180,E1 -24649.756,E2 -24649.756} C_VEL
LIN {X 0,Y 137.839,Z 389.119,A -85,B 0,C 180,E1 -24653.041,E2 -24653.041} C_VEL
LIN {X 0,Y 138.007,Z 379.707,A -85,B 0,C 180,E1 -24655.981,E2 -24655.981} C_VEL
LIN {X 0,Y 138.533,Z 369.156,A -85,B 0,C 180,E1 -24658.543,E2 -24658.543} C_VEL
LIN {X 0,Y 138.635,Z 363.538,A -85,B 0,C 180,E1 -24659.633,E2 -24659.633} C_VEL
LIN {X 0,Y 134.993,Z 340.585,A -85,B 0,C 180,E1 -24676.635,E2 -24676.635} C_VEL
LIN {X 0,Y 135.314,Z 332.336,A -85,B 0,C 180,E1 -24682.921,E2 -24682.921} C_VEL
LIN {X 0,Y 135.624,Z 327.593,A -85,B 0,C 180,E1 -24686.543,E2 -24686.543} C_VEL
LIN {X 0,Y 135.912,Z 327.558,A -85,B 0,C 180,E1 -24688.469,E2 -24688.469} C_VEL
LIN {X 0,Y 136.056,Z 327.538,A -85,B 0,C 180,E1 -24691.096,E2 -24691.096} C_VEL
LIN {X 0,Y 136.081,Z 327.527,A -85,B 0,C 180,E1 -24694.613,E2 -24694.613} C_VEL
LIN {X 0,Y 136.02,Z 327.542,A -85,B 0,C 180,E1 -24699.192,E2 -24699.192} C_VEL
LIN {X 0,Y 135.971,Z 327.544,A -85,B 0,C 180,E1 -24703.645,E2 -24703.645} C_VEL
LIN {X 0,Y 135.977,Z 327.546,A -85,B 0,C 180,E1 -24707.785,E2 -24707.785} C_VEL
LIN {X 0,Y 136.016,Z 327.536,A -85,B 0,C 180,E1 -24711.681,E2 -24711.681} C_VEL
LIN {X 0,Y 136.077,Z 327.534,A -85,B 0,C 180,E1 -24715.718,E2 -24715.718} C_VEL
LIN {X 0,Y 136.138,Z 327.525,A -85,B 0,C 180,E1 -24722.314,E2 -24722.314} C_VEL
LIN {X 0,Y 136.236,Z 327.509,A -85,B 0,C 180,E1 -24728.832,E2 -24728.832} C_VEL
LIN {X 0,Y 136.262,Z 327.509,A -85,B 0,C 180,E1 -24735.055,E2 -24735.055} C_VEL
LIN {X 0,Y 136.422,Z 327.486,A -85,B 0,C 180,E1 -24738.164,E2 -24738.164} C_VEL
LIN {X 0,Y 136.537,Z 327.477,A -85,B 0,C 180,E1 -24741.117,E2 -24741.117} C_VEL
LIN {X 0,Y 137.102,Z 327.408,A -85,B 0,C 180,E1 -24750,E2 -24750} C_VEL
LIN {X 0,Y 136.537,Z 327.477,A -85,B 0,C 180,E1 -24758.883,E2 -24758.883} C_VEL
LIN {X 0,Y 136.431,Z 327.485,A -85,B 0,C 180,E1 -24761.891,E2 -24761.891} C_VEL
LIN {X 0,Y 136.254,Z 327.512,A -85,B 0,C 180,E1 -24768.028,E2 -24768.028} C_VEL
LIN {X 0,Y 136.218,Z 327.512,A -85,B 0,C 180,E1 -24771.781,E2 -24771.781} C_VEL
LIN {X 0,Y 136.092,Z 327.529,A -85,B 0,C 180,E1 -24778.619,E2 -24778.619} C_VEL
LIN {X 0,Y 136.063,Z 327.536,A -85,B 0,C 180,E1 -24784.623,E2 -24784.623} C_VEL
LIN {X 0,Y 136.02,Z 327.536,A -85,B 0,C 180,E1 -24789.199,E2 -24789.199} C_VEL
LIN {X 0,Y 135.972,Z 327.547,A -85,B 0,C 180,E1 -24793.652,E2 -24793.652} C_VEL
